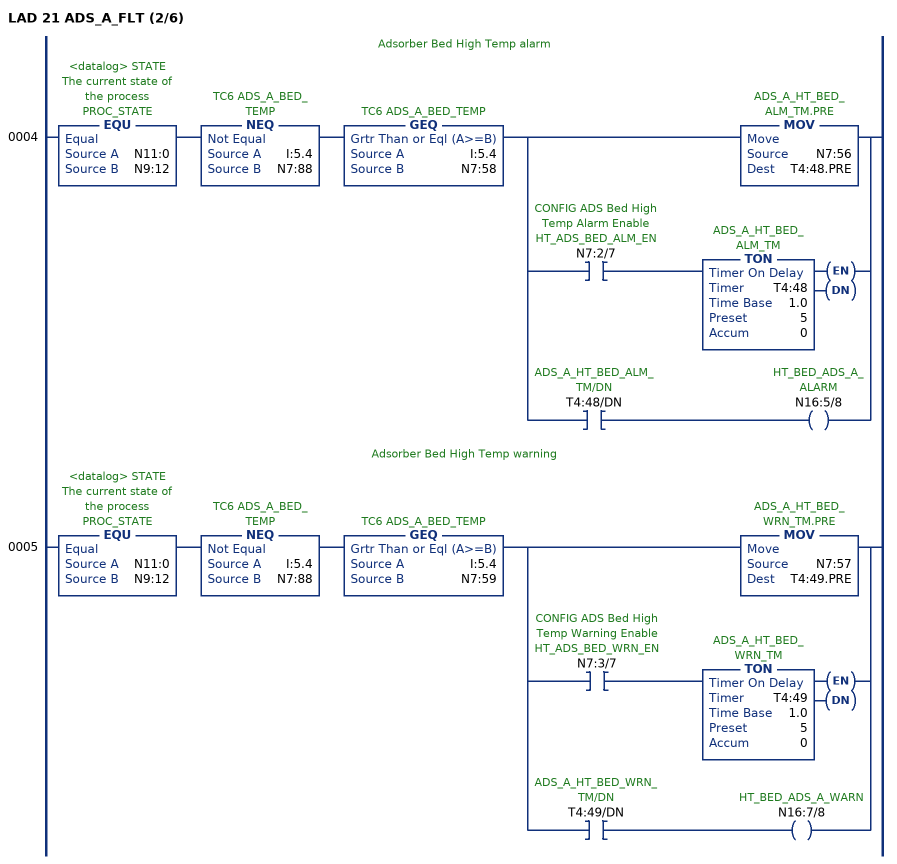
% Rung: 4 %
% Adsorber Bed High Temp alarm %
SOR EQU N11:0 N9:12 NEQ I:5.4 N7:88 GEQ I:5.4 N7:58 BST MOV N7:56 T4:48.PRE NXB XIC N7:2/7 TON T4:48 1.0 5 0 NXB XIC T4:48/DN OTE N16:5/8 BND EOR
%   N11:0  PROC_STATE  "<datalog> STATE The current state of the process" %
%   N9:12  PROC_REGEN_A  "STATE Process Regen A" %
%   I:5.4  ADS_A_BED_TEMP  "TC6" %
%   N7:88  TC_OPEN_SP  "CONFIG TC Open Setpoint" %
%   N7:58  HT_ADS_BED_ALM_SP  "CONFIG ADS Bed High Temp Alarm Setpoint" %
%   N7:56  HT_ADS_BED_ALM_DLY  "CONFIG ADS Bed High Temp Alarm Delay" %
%   T4:48  ADS_A_HT_BED_ALM_TM %
%   N7:2/7  HT_ADS_BED_ALM_EN  "CONFIG ADS Bed High Temp Alarm Enable" %
%   N16:5/8  HT_BED_ADS_A_ALARM %
% Rung: 5 %
% Adsorber Bed High Temp warning %
SOR EQU N11:0 N9:12 NEQ I:5.4 N7:88 GEQ I:5.4 N7:59 BST MOV N7:57 T4:49.PRE NXB XIC N7:3/7 TON T4:49 1.0 5 0 NXB XIC T4:49/DN OTE N16:7/8 BND EOR
%   N11:0  PROC_STATE  "<datalog> STATE The current state of the process" %
%   N9:12  PROC_REGEN_A  "STATE Process Regen A" %
%   I:5.4  ADS_A_BED_TEMP  "TC6" %
%   N7:88  TC_OPEN_SP  "CONFIG TC Open Setpoint" %
%   N7:59  HT_ADS_BED_WRN_SP  "CONFIG ADS Bed High Temp Warning Setpoint" %
%   N7:57  HT_ADS_BED_WRN_DLY  "CONFIG ADS Bed High Temp Warning Delay" %
%   T4:49  ADS_A_HT_BED_WRN_TM %
%   N7:3/7  HT_ADS_BED_WRN_EN  "CONFIG ADS Bed High Temp Warning Enable" %
%   N16:7/8  HT_BED_ADS_A_WARN %

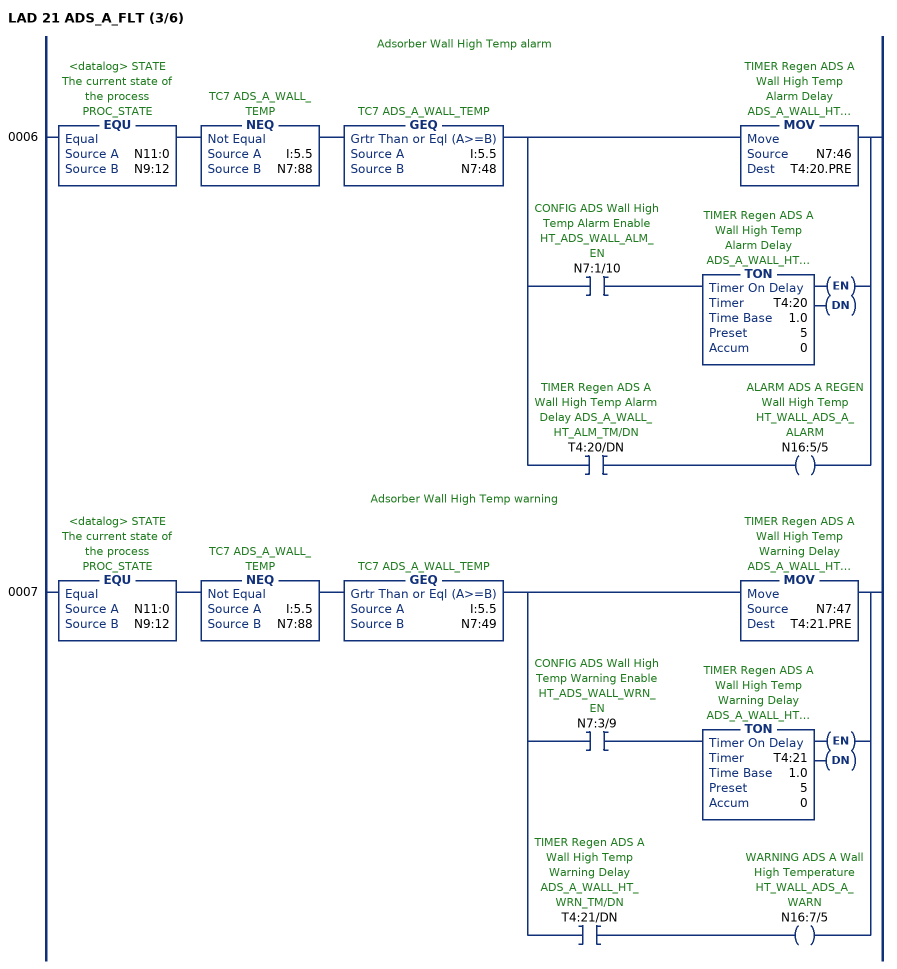
% Rung: 6 %
% Adsorber Wall High Temp alarm %
SOR EQU N11:0 N9:12 NEQ I:5.5 N7:88 GEQ I:5.5 N7:48 BST MOV N7:46 T4:20.PRE NXB XIC N7:1/10 TON T4:20 1.0 5 0 NXB XIC T4:20/DN OTE N16:5/5 BND EOR
%   N11:0  PROC_STATE  "<datalog> STATE The current state of the process" %
%   N9:12  PROC_REGEN_A  "STATE Process Regen A" %
%   I:5.5  ADS_A_WALL_TEMP  "TC7" %
%   N7:88  TC_OPEN_SP  "CONFIG TC Open Setpoint" %
%   N7:48  HT_ADS_WALL_ALM_SP  "CONFIG ADS Wall High Temp Alarm Setpoint" %
%   N7:46  HT_ADS_WALL_ALM_DLY  "CONFIG ADS Wall High Temp Alarm Delay" %
%   T4:20  ADS_A_WALL_HT_ALM_TM  "TIMER Regen ADS A Wall High Temp Alarm Delay" %
%   N7:1/10  HT_ADS_WALL_ALM_EN  "CONFIG ADS Wall High Temp Alarm Enable" %
%   N16:5/5  HT_WALL_ADS_A_ALARM  "ALARM ADS A REGEN Wall High Temp" %
% Rung: 7 %
% Adsorber Wall High Temp warning %
SOR EQU N11:0 N9:12 NEQ I:5.5 N7:88 GEQ I:5.5 N7:49 BST MOV N7:47 T4:21.PRE NXB XIC N7:3/9 TON T4:21 1.0 5 0 NXB XIC T4:21/DN OTE N16:7/5 BND EOR
%   N11:0  PROC_STATE  "<datalog> STATE The current state of the process" %
%   N9:12  PROC_REGEN_A  "STATE Process Regen A" %
%   I:5.5  ADS_A_WALL_TEMP  "TC7" %
%   N7:88  TC_OPEN_SP  "CONFIG TC Open Setpoint" %
%   N7:49  HT_ADS_WALL_WRN_SP  "CONFIG ADS Wall High Temp Warning Setpoint" %
%   N7:47  HT_ADS_WALL_WRN_DLY  "CONFIG ADS Wall High Temp Warning Delay" %
%   T4:21  ADS_A_WALL_HT_WRN_TM  "TIMER Regen ADS A Wall High Temp Warning Delay" %
%   N7:3/9  HT_ADS_WALL_WRN_EN  "CONFIG ADS Wall High Temp Warning Enable" %
%   N16:7/5  HT_WALL_ADS_A_WARN  "WARNING ADS A Wall High Temperature" %

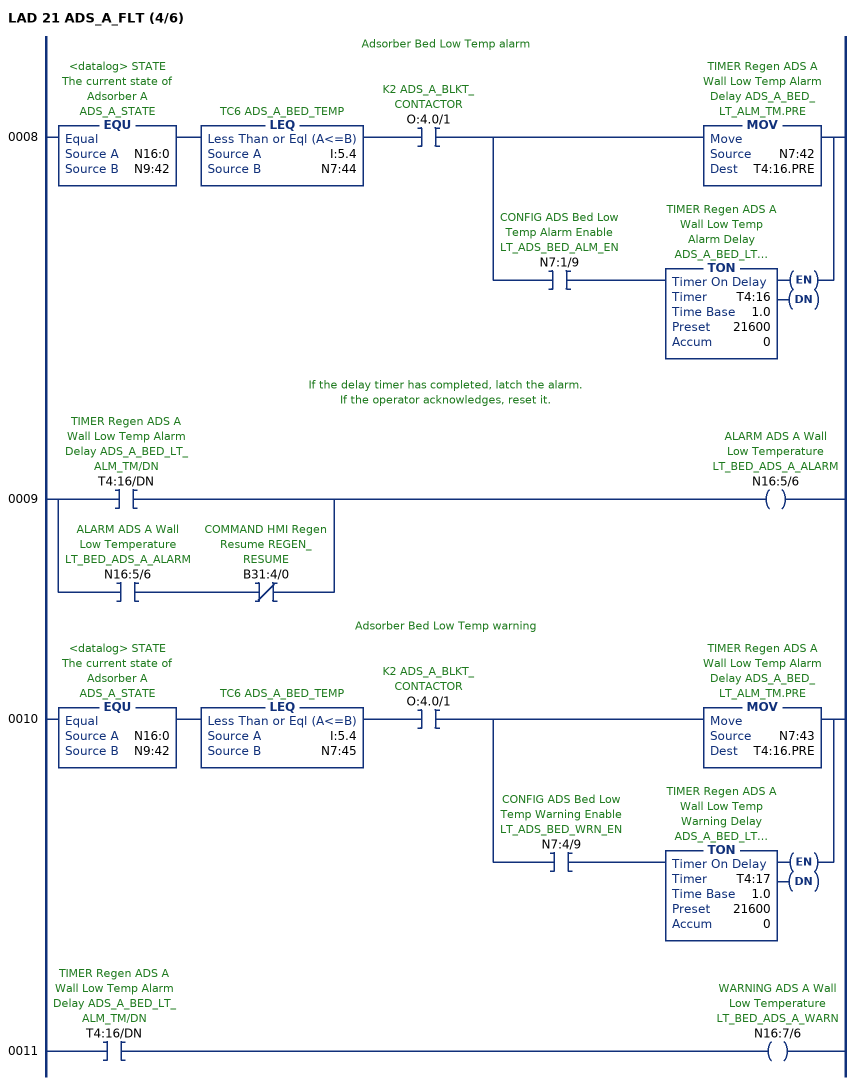
% Rung: 8 %
% Adsorber Bed Low Temp alarm %
SOR EQU N16:0 N9:42 LEQ I:5.4 N7:44 XIC O:4.0/1 BST MOV N7:42 T4:16.PRE NXB XIC N7:1/9 TON T4:16 1.0 21600 0 BND EOR
%   N16:0  ADS_A_STATE  "<datalog> STATE The current state of Adsorber A" %
%   N9:42  ADS_REGEN  "STATE ADS Regen" %
%   I:5.4  ADS_A_BED_TEMP  "TC6" %
%   N7:44  LT_ADS_BED_ALM_SP  "CONFIG ADS Bed Low Temp Alarm Setpoint" %
%   O:4.0/1  ADS_A_BLKT_CONTACTOR  "K2" %
%   N7:42  LT_ADS_BED_ALM_DLY  "CONFIG ADS Bed Low Temp Alarm Delay" %
%   T4:16  ADS_A_BED_LT_ALM_TM  "TIMER Regen ADS A Wall Low Temp Alarm Delay" %
%   N7:1/9  LT_ADS_BED_ALM_EN  "CONFIG ADS Bed Low Temp Alarm Enable" %
% Rung: 9 %
% If the delay timer has completed, latch the alarm.
% If the operator acknowledges, reset it. %
SOR BST XIC T4:16/DN NXB XIC N16:5/6 XIO B31:4/0 BND OTE N16:5/6 EOR
%   T4:16  ADS_A_BED_LT_ALM_TM  "TIMER Regen ADS A Wall Low Temp Alarm Delay" %
%   N16:5/6  LT_BED_ADS_A_ALARM  "ALARM ADS A Wall Low Temperature" %
%   B31:4/0  REGEN_RESUME  "COMMAND HMI Regen Resume" %
% Rung: 10 %
% Adsorber Bed Low Temp warning %
SOR EQU N16:0 N9:42 LEQ I:5.4 N7:45 XIC O:4.0/1 BST MOV N7:43 T4:16.PRE NXB XIC N7:4/9 TON T4:17 1.0 21600 0 BND EOR
%   N16:0  ADS_A_STATE  "<datalog> STATE The current state of Adsorber A" %
%   N9:42  ADS_REGEN  "STATE ADS Regen" %
%   I:5.4  ADS_A_BED_TEMP  "TC6" %
%   N7:45  LT_ADS_BED_WRN_SP  "CONFIG ADS Bed Low Temp Warning Setpoint" %
%   O:4.0/1  ADS_A_BLKT_CONTACTOR  "K2" %
%   N7:43  LT_ADS_BED_WRN_DLY  "CONFIG ADS Bed Low Temp Warning Delay" %
%   T4:16  ADS_A_BED_LT_ALM_TM  "TIMER Regen ADS A Wall Low Temp Alarm Delay" %
%   N7:4/9  LT_ADS_BED_WRN_EN  "CONFIG ADS Bed Low Temp Warning Enable" %
%   T4:17  ADS_A_BED_LT_WRN_TM  "TIMER Regen ADS A Wall Low Temp Warning Delay" %
% Rung: 11 %
SOR XIC T4:16/DN OTE N16:7/6 EOR
%   T4:16  ADS_A_BED_LT_ALM_TM  "TIMER Regen ADS A Wall Low Temp Alarm Delay" %
%   N16:7/6  LT_BED_ADS_A_WARN  "WARNING ADS A Wall Low Temperature" %

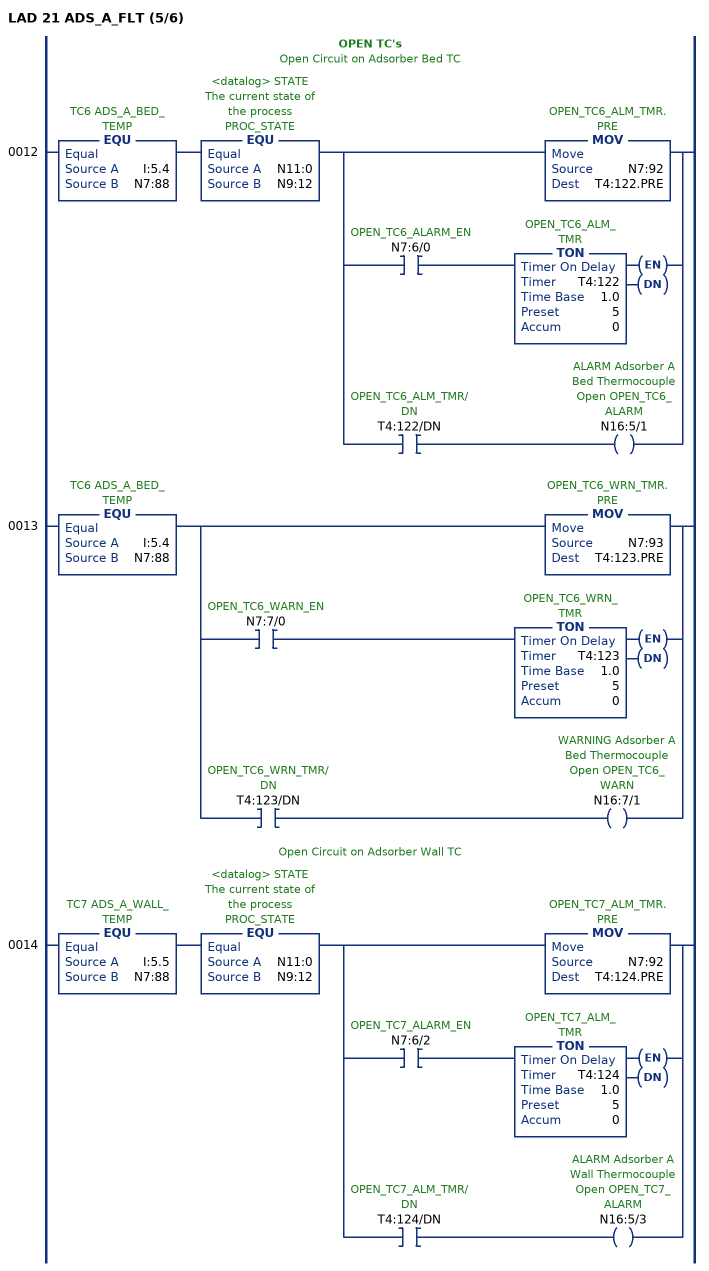
% Rung: 12 %
% TITLE: OPEN TC's %
% Open Circuit on Adsorber Bed TC %
SOR EQU I:5.4 N7:88 EQU N11:0 N9:12 BST MOV N7:92 T4:122.PRE NXB XIC N7:6/0 TON T4:122 1.0 5 0 NXB XIC T4:122/DN OTE N16:5/1 BND EOR
%   I:5.4  ADS_A_BED_TEMP  "TC6" %
%   N7:88  TC_OPEN_SP  "CONFIG TC Open Setpoint" %
%   N11:0  PROC_STATE  "<datalog> STATE The current state of the process" %
%   N9:12  PROC_REGEN_A  "STATE Process Regen A" %
%   N7:92  OPEN_TC_ALM_DLY  "CONFIG TC Open Alarm Delay" %
%   T4:122  OPEN_TC6_ALM_TMR %
%   N7:6/0  OPEN_TC6_ALARM_EN %
%   N16:5/1  OPEN_TC6_ALARM  "ALARM Adsorber A Bed Thermocouple Open" %
% Rung: 13 %
SOR EQU I:5.4 N7:88 BST MOV N7:93 T4:123.PRE NXB XIC N7:7/0 TON T4:123 1.0 5 0 NXB XIC T4:123/DN OTE N16:7/1 BND EOR
%   I:5.4  ADS_A_BED_TEMP  "TC6" %
%   N7:88  TC_OPEN_SP  "CONFIG TC Open Setpoint" %
%   N7:93  OPEN_TC_WRN_DLY  "CONFIG TC Open Warning Delay" %
%   T4:123  OPEN_TC6_WRN_TMR %
%   N7:7/0  OPEN_TC6_WARN_EN %
%   N16:7/1  OPEN_TC6_WARN  "WARNING Adsorber A Bed Thermocouple Open" %
% Rung: 14 %
% Open Circuit on Adsorber Wall TC %
SOR EQU I:5.5 N7:88 EQU N11:0 N9:12 BST MOV N7:92 T4:124.PRE NXB XIC N7:6/2 TON T4:124 1.0 5 0 NXB XIC T4:124/DN OTE N16:5/3 BND EOR
%   I:5.5  ADS_A_WALL_TEMP  "TC7" %
%   N7:88  TC_OPEN_SP  "CONFIG TC Open Setpoint" %
%   N11:0  PROC_STATE  "<datalog> STATE The current state of the process" %
%   N9:12  PROC_REGEN_A  "STATE Process Regen A" %
%   N7:92  OPEN_TC_ALM_DLY  "CONFIG TC Open Alarm Delay" %
%   T4:124  OPEN_TC7_ALM_TMR %
%   N7:6/2  OPEN_TC7_ALARM_EN %
%   N16:5/3  OPEN_TC7_ALARM  "ALARM Adsorber A Wall Thermocouple Open" %

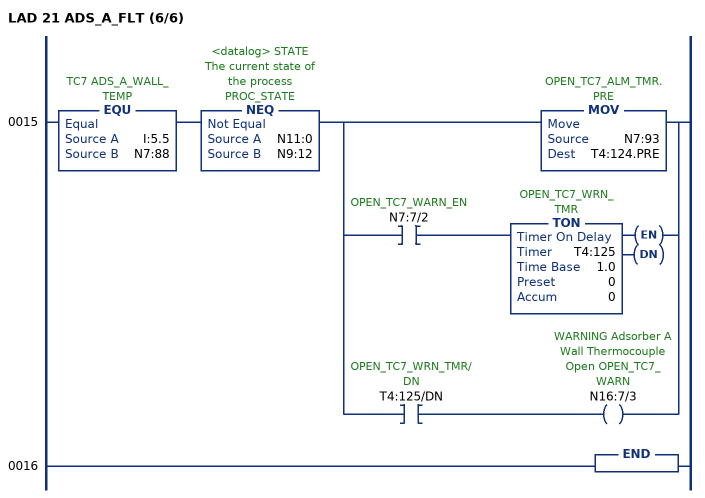
% Rung: 15 %
SOR EQU I:5.5 N7:88 NEQ N11:0 N9:12 BST MOV N7:93 T4:124.PRE NXB XIC N7:7/2 TON T4:125 1.0 0 0 NXB XIC T4:125/DN OTE N16:7/3 BND EOR
%   I:5.5  ADS_A_WALL_TEMP  "TC7" %
%   N7:88  TC_OPEN_SP  "CONFIG TC Open Setpoint" %
%   N11:0  PROC_STATE  "<datalog> STATE The current state of the process" %
%   N9:12  PROC_REGEN_A  "STATE Process Regen A" %
%   N7:93  OPEN_TC_WRN_DLY  "CONFIG TC Open Warning Delay" %
%   T4:124  OPEN_TC7_ALM_TMR %
%   N7:7/2  OPEN_TC7_WARN_EN %
%   T4:125  OPEN_TC7_WRN_TMR %
%   N16:7/3  OPEN_TC7_WARN  "WARNING Adsorber A Wall Thermocouple Open" %
% Rung: 16 %
SOR END EOR

LADDER 22 "ADS_B"    % Controld Adsorber B %
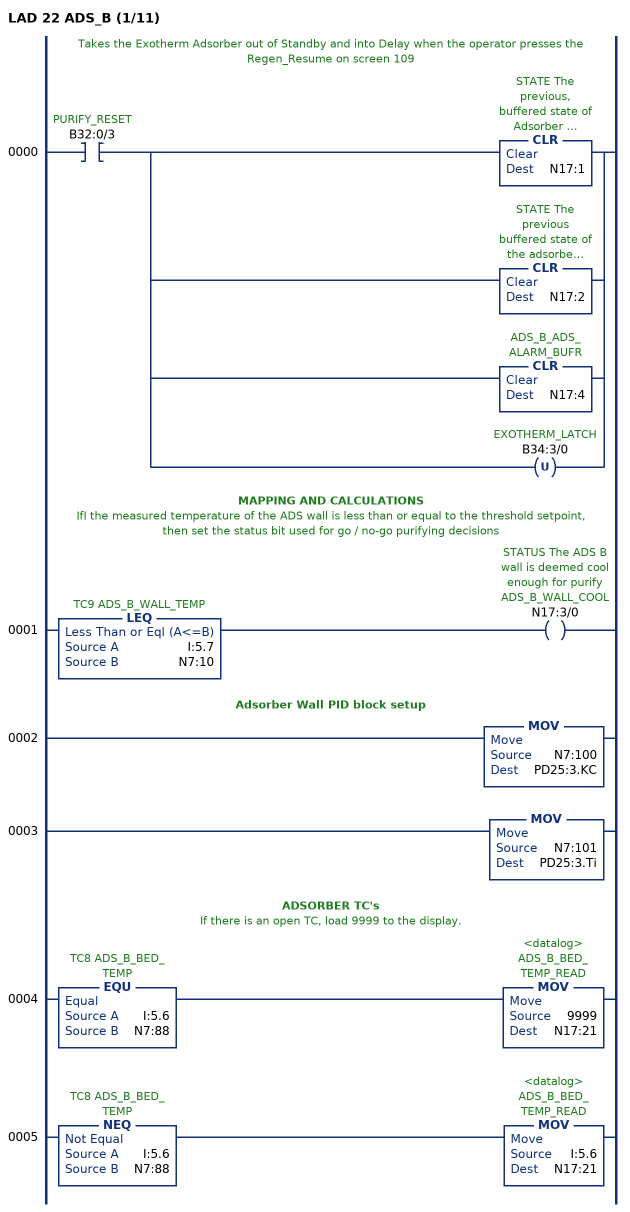
% Rung: 0 %
% Takes the Exotherm Adsorber out of Standby and into Delay when the operator presses the Regen_Resume on screen 109 %
SOR XIC B32:0/3 BST CLR N17:1 NXB CLR N17:2 NXB CLR N17:4 NXB OTU B34:3/0 BND EOR
%   B32:0/3  PURIFY_RESET %
%   N17:1  ADS_B_STANDBY_BUFFER  "STATE The previous, buffered state of Adsorber B" %
%   N17:2  ADS_B_SYS_ALARM_BUFR  "STATE The previous buffered state of the adsorber when the alarm occured" %
%   N17:4  ADS_B_ADS_ALARM_BUFR %
%   B34:3/0  EXOTHERM_LATCH %
% Rung: 1 %
% TITLE: MAPPING AND CALCULATIONS %
% IfI the measured temperature of the ADS wall is less than or equal to the threshold setpoint, then set the status bit used for go / no-go purifying decisions %
SOR LEQ I:5.7 N7:10 OTE N17:3/0 EOR
%   I:5.7  ADS_B_WALL_TEMP  "TC9" %
%   N7:10  ADS_WALL_TEMP_COOL  "CONFIG The temp at which the adsorber wall is deemed to be cool enough to purify" %
%   N17:3/0  ADS_B_WALL_COOL  "STATUS The ADS B wall is deemed cool enough for purify" %
% Rung: 2 %
% TITLE: Adsorber Wall PID block setup %
SOR MOV N7:100 PD25:3.KC EOR
%   N7:100  BLANKET_P  "CONFIG Blanket Proportional Gain" %
% Rung: 3 %
SOR MOV N7:101 PD25:3.Ti EOR
%   N7:101  BLANKET_I  "CONFIG Blanket Integral Gain" %
% Rung: 4 %
% TITLE: ADSORBER TC's %
% If there is an open TC, load 9999 to the display. %
SOR EQU I:5.6 N7:88 MOV 9999 N17:21 EOR
%   I:5.6  ADS_B_BED_TEMP  "TC8" %
%   N7:88  TC_OPEN_SP  "CONFIG TC Open Setpoint" %
%   N17:21  ADS_B_BED_TEMP_READ  "<datalog>" %
% Rung: 5 %
SOR NEQ I:5.6 N7:88 MOV I:5.6 N17:21 EOR
%   I:5.6  ADS_B_BED_TEMP  "TC8" %
%   N7:88  TC_OPEN_SP  "CONFIG TC Open Setpoint" %
%   N17:21  ADS_B_BED_TEMP_READ  "<datalog>" %

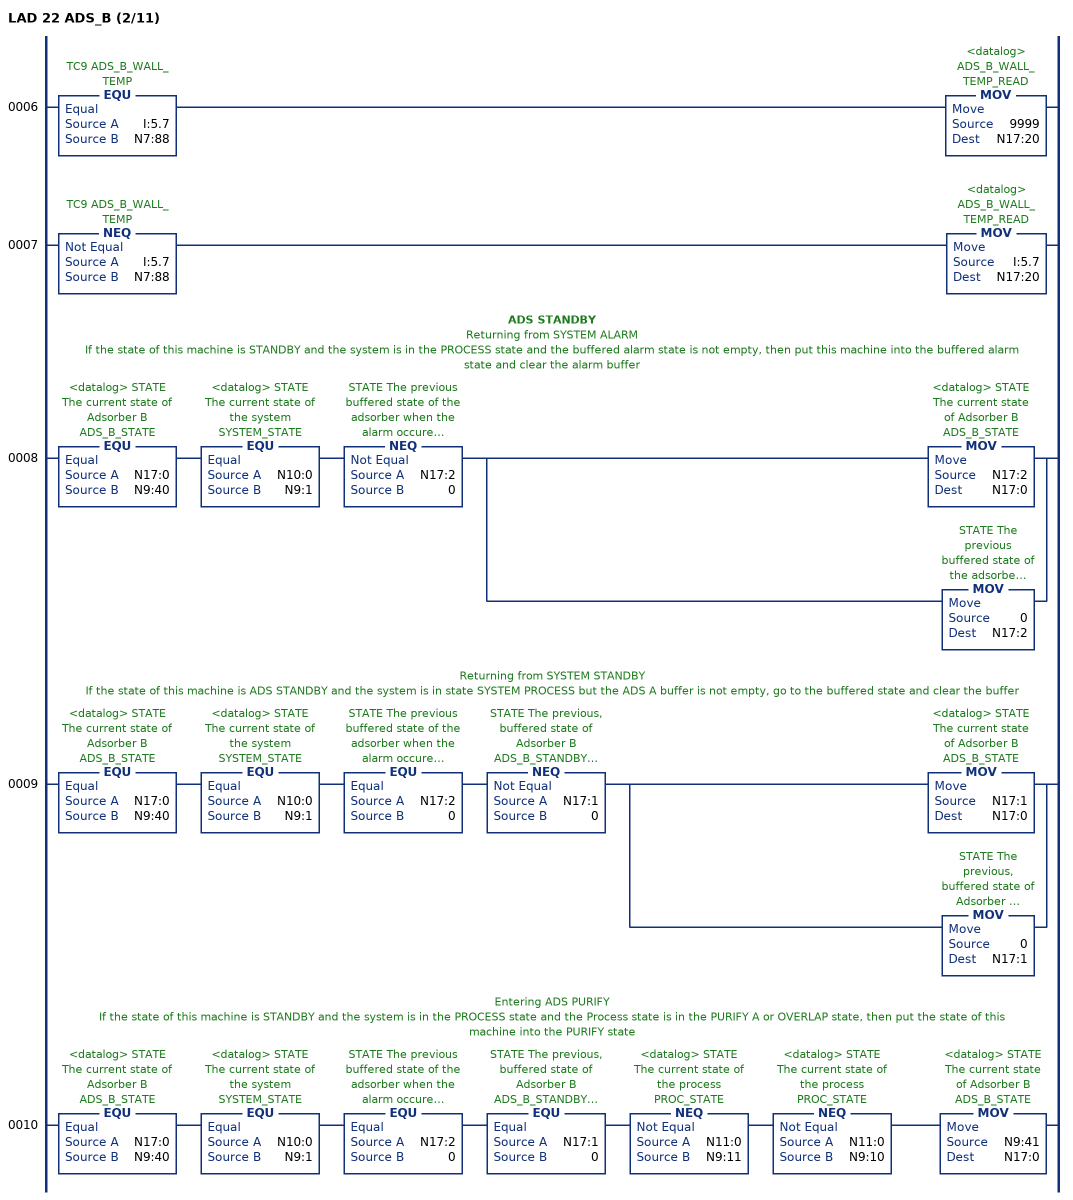
% Rung: 6 %
SOR EQU I:5.7 N7:88 MOV 9999 N17:20 EOR
%   I:5.7  ADS_B_WALL_TEMP  "TC9" %
%   N7:88  TC_OPEN_SP  "CONFIG TC Open Setpoint" %
%   N17:20  ADS_B_WALL_TEMP_READ  "<datalog>" %
% Rung: 7 %
SOR NEQ I:5.7 N7:88 MOV I:5.7 N17:20 EOR
%   I:5.7  ADS_B_WALL_TEMP  "TC9" %
%   N7:88  TC_OPEN_SP  "CONFIG TC Open Setpoint" %
%   N17:20  ADS_B_WALL_TEMP_READ  "<datalog>" %
% Rung: 8 %
% TITLE: ADS STANDBY %
% Returning from SYSTEM ALARM
% If the state of this machine is STANDBY and the system is in the PROCESS state and the buffered alarm state is not empty, then put this machine into the buffered alarm state and clear the alarm buffer %
SOR EQU N17:0 N9:40 EQU N10:0 N9:1 NEQ N17:2 0 BST MOV N17:2 N17:0 NXB MOV 0 N17:2 BND EOR
%   N17:0  ADS_B_STATE  "<datalog> STATE The current state of Adsorber B" %
%   N9:40  ADS_STANDBY  "STATE ADS Standby" %
%   N10:0  SYSTEM_STATE  "<datalog> STATE The current state of the system" %
%   N9:1  SYSTEM_PROCESS  "STATE System Process" %
%   N17:2  ADS_B_SYS_ALARM_BUFR  "STATE The previous buffered state of the adsorber when the alarm occured" %
% Rung: 9 %
% Returning from SYSTEM STANDBY
% If the state of this machine is ADS STANDBY and the system is in state SYSTEM PROCESS but the ADS A buffer is not empty, go to the buffered state and clear the buffer %
SOR EQU N17:0 N9:40 EQU N10:0 N9:1 EQU N17:2 0 NEQ N17:1 0 BST MOV N17:1 N17:0 NXB MOV 0 N17:1 BND EOR
%   N17:0  ADS_B_STATE  "<datalog> STATE The current state of Adsorber B" %
%   N9:40  ADS_STANDBY  "STATE ADS Standby" %
%   N10:0  SYSTEM_STATE  "<datalog> STATE The current state of the system" %
%   N9:1  SYSTEM_PROCESS  "STATE System Process" %
%   N17:2  ADS_B_SYS_ALARM_BUFR  "STATE The previous buffered state of the adsorber when the alarm occured" %
%   N17:1  ADS_B_STANDBY_BUFFER  "STATE The previous, buffered state of Adsorber B" %
% Rung: 10 %
% Entering ADS PURIFY
% If the state of this machine is STANDBY and the system is in the PROCESS state and the Process state is in the PURIFY A or OVERLAP state, then put the state of this machine into the PURIFY state %
SOR EQU N17:0 N9:40 EQU N10:0 N9:1 EQU N17:2 0 EQU N17:1 0 NEQ N11:0 N9:11 NEQ N11:0 N9:10 MOV N9:41 N17:0 EOR
%   N17:0  ADS_B_STATE  "<datalog> STATE The current state of Adsorber B" %
%   N9:40  ADS_STANDBY  "STATE ADS Standby" %
%   N10:0  SYSTEM_STATE  "<datalog> STATE The current state of the system" %
%   N9:1  SYSTEM_PROCESS  "STATE System Process" %
%   N17:2  ADS_B_SYS_ALARM_BUFR  "STATE The previous buffered state of the adsorber when the alarm occured" %
%   N17:1  ADS_B_STANDBY_BUFFER  "STATE The previous, buffered state of Adsorber B" %
%   N11:0  PROC_STATE  "<datalog> STATE The current state of the process" %
%   N9:11  PROC_REGEN_B  "STATE Process Regen B" %
%   N9:10  PROCESS_STANDBY  "STATE Process Standby" %
%   N9:41  ADS_PURIFY  "STATE ADS Purify" %

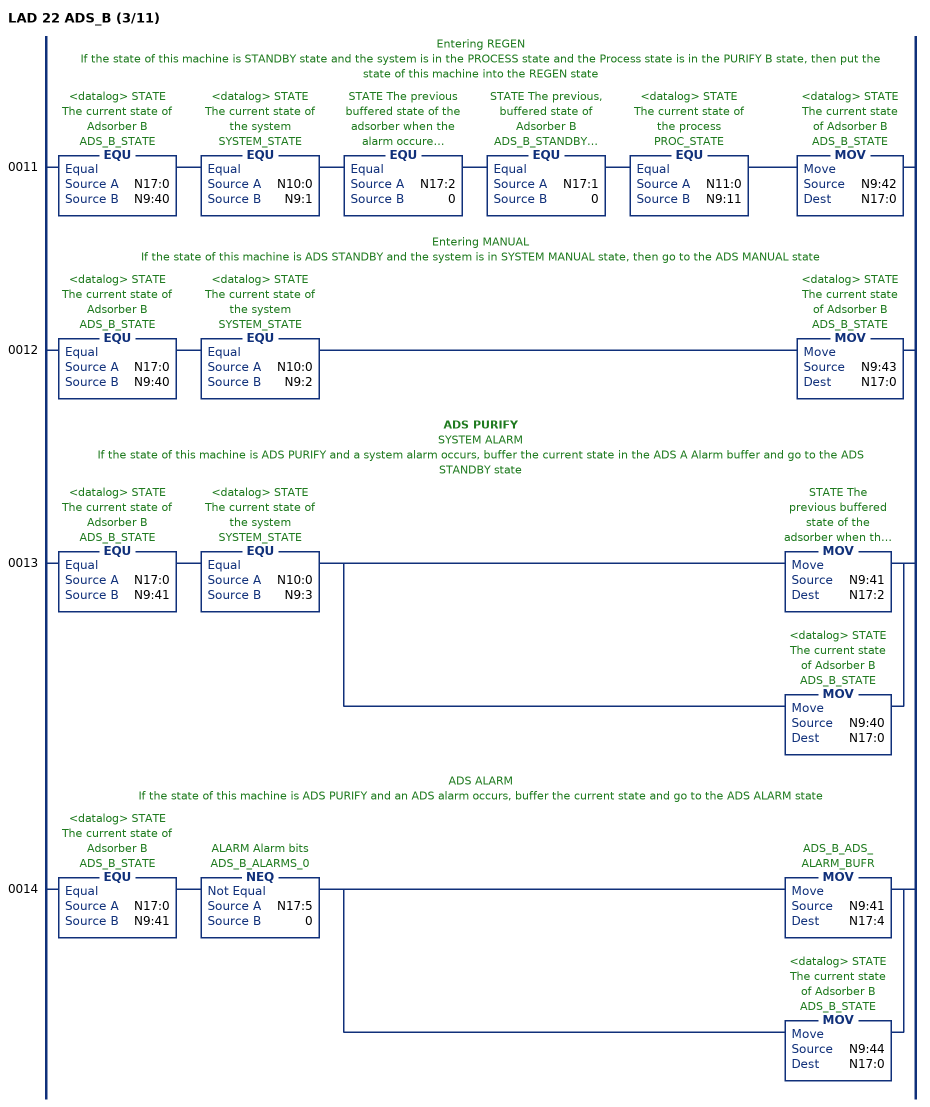
% Rung: 11 %
% Entering REGEN
% If the state of this machine is STANDBY state and the system is in the PROCESS state and the Process state is in the PURIFY B state, then put the state of this machine into the REGEN state %
SOR EQU N17:0 N9:40 EQU N10:0 N9:1 EQU N17:2 0 EQU N17:1 0 EQU N11:0 N9:11 MOV N9:42 N17:0 EOR
%   N17:0  ADS_B_STATE  "<datalog> STATE The current state of Adsorber B" %
%   N9:40  ADS_STANDBY  "STATE ADS Standby" %
%   N10:0  SYSTEM_STATE  "<datalog> STATE The current state of the system" %
%   N9:1  SYSTEM_PROCESS  "STATE System Process" %
%   N17:2  ADS_B_SYS_ALARM_BUFR  "STATE The previous buffered state of the adsorber when the alarm occured" %
%   N17:1  ADS_B_STANDBY_BUFFER  "STATE The previous, buffered state of Adsorber B" %
%   N11:0  PROC_STATE  "<datalog> STATE The current state of the process" %
%   N9:11  PROC_REGEN_B  "STATE Process Regen B" %
%   N9:42  ADS_REGEN  "STATE ADS Regen" %
% Rung: 12 %
% Entering MANUAL
% If the state of this machine is ADS STANDBY and the system is in SYSTEM MANUAL state, then go to the ADS MANUAL state %
SOR EQU N17:0 N9:40 EQU N10:0 N9:2 MOV N9:43 N17:0 EOR
%   N17:0  ADS_B_STATE  "<datalog> STATE The current state of Adsorber B" %
%   N9:40  ADS_STANDBY  "STATE ADS Standby" %
%   N10:0  SYSTEM_STATE  "<datalog> STATE The current state of the system" %
%   N9:2  SYSTEM_MANUAL  "STATE System Manual" %
%   N9:43  ADS_MANUAL  "STATE ADS Manual" %
% Rung: 13 %
% TITLE: ADS PURIFY %
% SYSTEM ALARM
% If the state of this machine is ADS PURIFY and a system alarm occurs, buffer the current state in the ADS A Alarm buffer and go to the ADS STANDBY state %
SOR EQU N17:0 N9:41 EQU N10:0 N9:3 BST MOV N9:41 N17:2 NXB MOV N9:40 N17:0 BND EOR
%   N17:0  ADS_B_STATE  "<datalog> STATE The current state of Adsorber B" %
%   N9:41  ADS_PURIFY  "STATE ADS Purify" %
%   N10:0  SYSTEM_STATE  "<datalog> STATE The current state of the system" %
%   N9:3  SYSTEM_ALARM  "STATE System Alarm" %
%   N17:2  ADS_B_SYS_ALARM_BUFR  "STATE The previous buffered state of the adsorber when the alarm occured" %
%   N9:40  ADS_STANDBY  "STATE ADS Standby" %
% Rung: 14 %
% ADS ALARM
% If the state of this machine is ADS PURIFY and an ADS alarm occurs, buffer the current state and go to the ADS ALARM state %
SOR EQU N17:0 N9:41 NEQ N17:5 0 BST MOV N9:41 N17:4 NXB MOV N9:44 N17:0 BND EOR
%   N17:0  ADS_B_STATE  "<datalog> STATE The current state of Adsorber B" %
%   N9:41  ADS_PURIFY  "STATE ADS Purify" %
%   N17:5  ADS_B_ALARMS_0  "ALARM Alarm bits" %
%   N17:4  ADS_B_ADS_ALARM_BUFR %
%   N9:44  ADS_ALARM  "STATE ADS Alarm" %

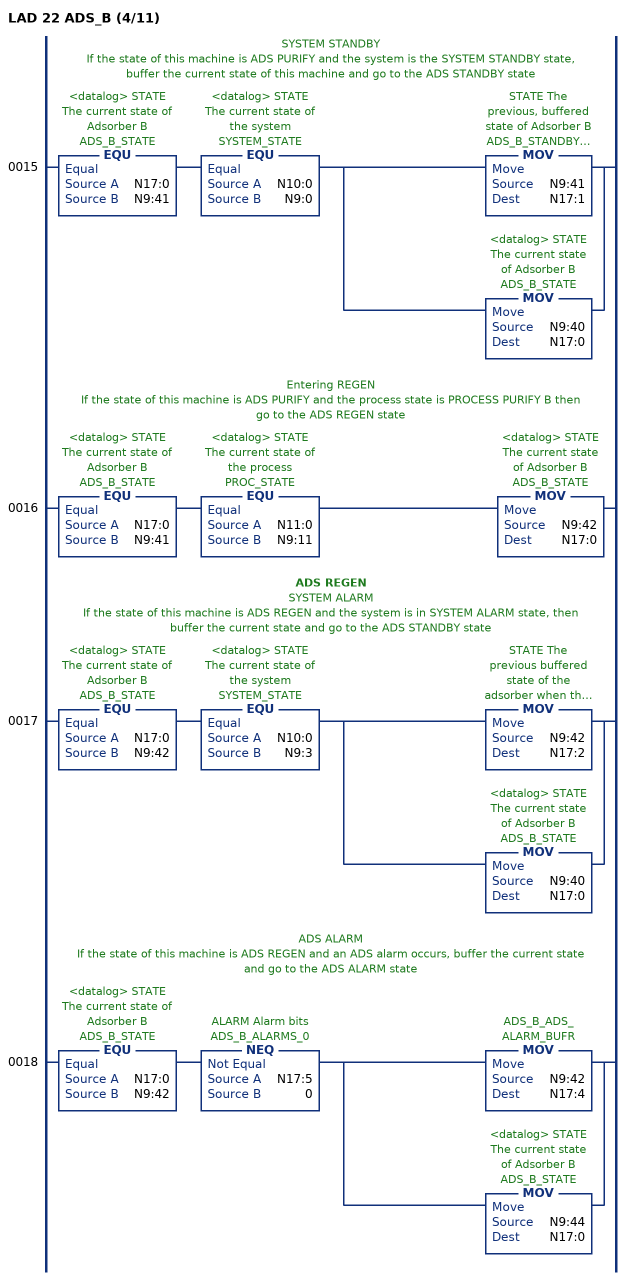
% Rung: 15 %
% SYSTEM STANDBY
% If the state of this machine is ADS PURIFY and the system is the SYSTEM STANDBY state, buffer the current state of this machine and go to the ADS STANDBY state %
SOR EQU N17:0 N9:41 EQU N10:0 N9:0 BST MOV N9:41 N17:1 NXB MOV N9:40 N17:0 BND EOR
%   N17:0  ADS_B_STATE  "<datalog> STATE The current state of Adsorber B" %
%   N9:41  ADS_PURIFY  "STATE ADS Purify" %
%   N10:0  SYSTEM_STATE  "<datalog> STATE The current state of the system" %
%   N9:0  SYSTEM_STANDBY  "STATE System Standby" %
%   N17:1  ADS_B_STANDBY_BUFFER  "STATE The previous, buffered state of Adsorber B" %
%   N9:40  ADS_STANDBY  "STATE ADS Standby" %
% Rung: 16 %
% Entering REGEN
% If the state of this machine is ADS PURIFY and the process state is PROCESS PURIFY B then go to the ADS REGEN state %
SOR EQU N17:0 N9:41 EQU N11:0 N9:11 MOV N9:42 N17:0 EOR
%   N17:0  ADS_B_STATE  "<datalog> STATE The current state of Adsorber B" %
%   N9:41  ADS_PURIFY  "STATE ADS Purify" %
%   N11:0  PROC_STATE  "<datalog> STATE The current state of the process" %
%   N9:11  PROC_REGEN_B  "STATE Process Regen B" %
%   N9:42  ADS_REGEN  "STATE ADS Regen" %
% Rung: 17 %
% TITLE: ADS REGEN %
% SYSTEM ALARM
% If the state of this machine is ADS REGEN and the system is in SYSTEM ALARM state, then buffer the current state and go to the ADS STANDBY state %
SOR EQU N17:0 N9:42 EQU N10:0 N9:3 BST MOV N9:42 N17:2 NXB MOV N9:40 N17:0 BND EOR
%   N17:0  ADS_B_STATE  "<datalog> STATE The current state of Adsorber B" %
%   N9:42  ADS_REGEN  "STATE ADS Regen" %
%   N10:0  SYSTEM_STATE  "<datalog> STATE The current state of the system" %
%   N9:3  SYSTEM_ALARM  "STATE System Alarm" %
%   N17:2  ADS_B_SYS_ALARM_BUFR  "STATE The previous buffered state of the adsorber when the alarm occured" %
%   N9:40  ADS_STANDBY  "STATE ADS Standby" %
% Rung: 18 %
% ADS ALARM
% If the state of this machine is ADS REGEN and an ADS alarm occurs, buffer the current state and go to the ADS ALARM state %
SOR EQU N17:0 N9:42 NEQ N17:5 0 BST MOV N9:42 N17:4 NXB MOV N9:44 N17:0 BND EOR
%   N17:0  ADS_B_STATE  "<datalog> STATE The current state of Adsorber B" %
%   N9:42  ADS_REGEN  "STATE ADS Regen" %
%   N17:5  ADS_B_ALARMS_0  "ALARM Alarm bits" %
%   N17:4  ADS_B_ADS_ALARM_BUFR %
%   N9:44  ADS_ALARM  "STATE ADS Alarm" %

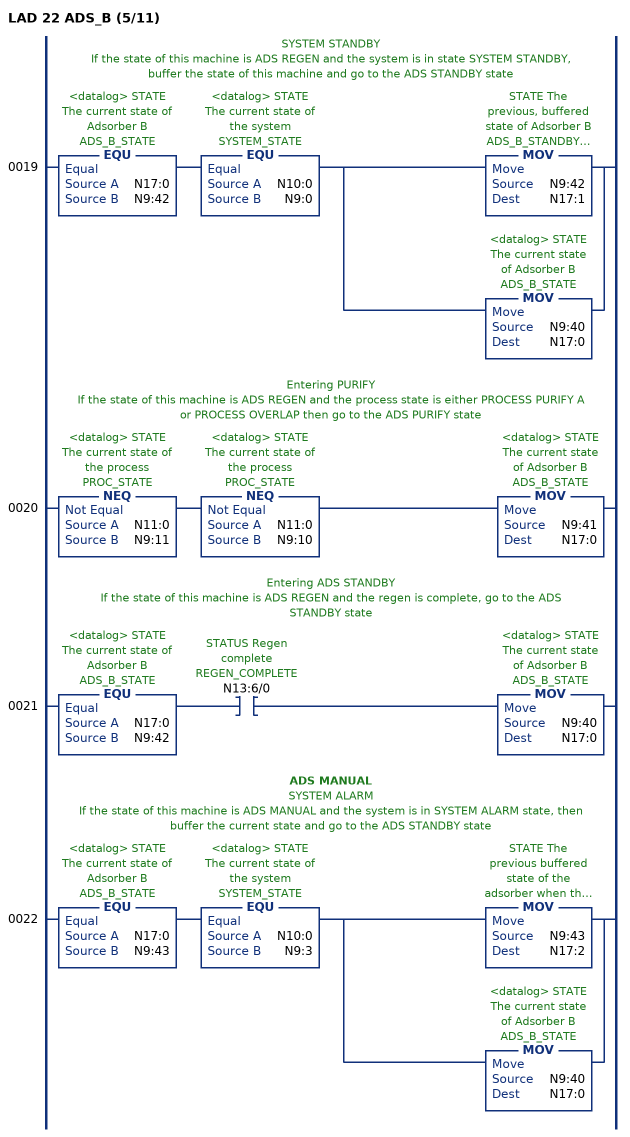
% Rung: 19 %
% SYSTEM STANDBY
% If the state of this machine is ADS REGEN and the system is in state SYSTEM STANDBY, buffer the state of this machine and go to the ADS STANDBY state %
SOR EQU N17:0 N9:42 EQU N10:0 N9:0 BST MOV N9:42 N17:1 NXB MOV N9:40 N17:0 BND EOR
%   N17:0  ADS_B_STATE  "<datalog> STATE The current state of Adsorber B" %
%   N9:42  ADS_REGEN  "STATE ADS Regen" %
%   N10:0  SYSTEM_STATE  "<datalog> STATE The current state of the system" %
%   N9:0  SYSTEM_STANDBY  "STATE System Standby" %
%   N17:1  ADS_B_STANDBY_BUFFER  "STATE The previous, buffered state of Adsorber B" %
%   N9:40  ADS_STANDBY  "STATE ADS Standby" %
% Rung: 20 %
% Entering PURIFY
% If the state of this machine is ADS REGEN and the process state is either PROCESS PURIFY A or PROCESS OVERLAP then go to the ADS PURIFY state %
SOR NEQ N11:0 N9:11 NEQ N11:0 N9:10 MOV N9:41 N17:0 EOR
%   N11:0  PROC_STATE  "<datalog> STATE The current state of the process" %
%   N9:11  PROC_REGEN_B  "STATE Process Regen B" %
%   N9:10  PROCESS_STANDBY  "STATE Process Standby" %
%   N9:41  ADS_PURIFY  "STATE ADS Purify" %
%   N17:0  ADS_B_STATE  "<datalog> STATE The current state of Adsorber B" %
% Rung: 21 %
% Entering ADS STANDBY
% If the state of this machine is ADS REGEN and the regen is complete, go to the ADS STANDBY state %
SOR EQU N17:0 N9:42 XIC N13:6/0 MOV N9:40 N17:0 EOR
%   N17:0  ADS_B_STATE  "<datalog> STATE The current state of Adsorber B" %
%   N9:42  ADS_REGEN  "STATE ADS Regen" %
%   N13:6/0  REGEN_COMPLETE  "STATUS Regen complete" %
%   N9:40  ADS_STANDBY  "STATE ADS Standby" %
% Rung: 22 %
% TITLE: ADS MANUAL %
% SYSTEM ALARM
% If the state of this machine is ADS MANUAL and the system is in SYSTEM ALARM state, then buffer the current state and go to the ADS STANDBY state %
SOR EQU N17:0 N9:43 EQU N10:0 N9:3 BST MOV N9:43 N17:2 NXB MOV N9:40 N17:0 BND EOR
%   N17:0  ADS_B_STATE  "<datalog> STATE The current state of Adsorber B" %
%   N9:43  ADS_MANUAL  "STATE ADS Manual" %
%   N10:0  SYSTEM_STATE  "<datalog> STATE The current state of the system" %
%   N9:3  SYSTEM_ALARM  "STATE System Alarm" %
%   N17:2  ADS_B_SYS_ALARM_BUFR  "STATE The previous buffered state of the adsorber when the alarm occured" %
%   N9:40  ADS_STANDBY  "STATE ADS Standby" %

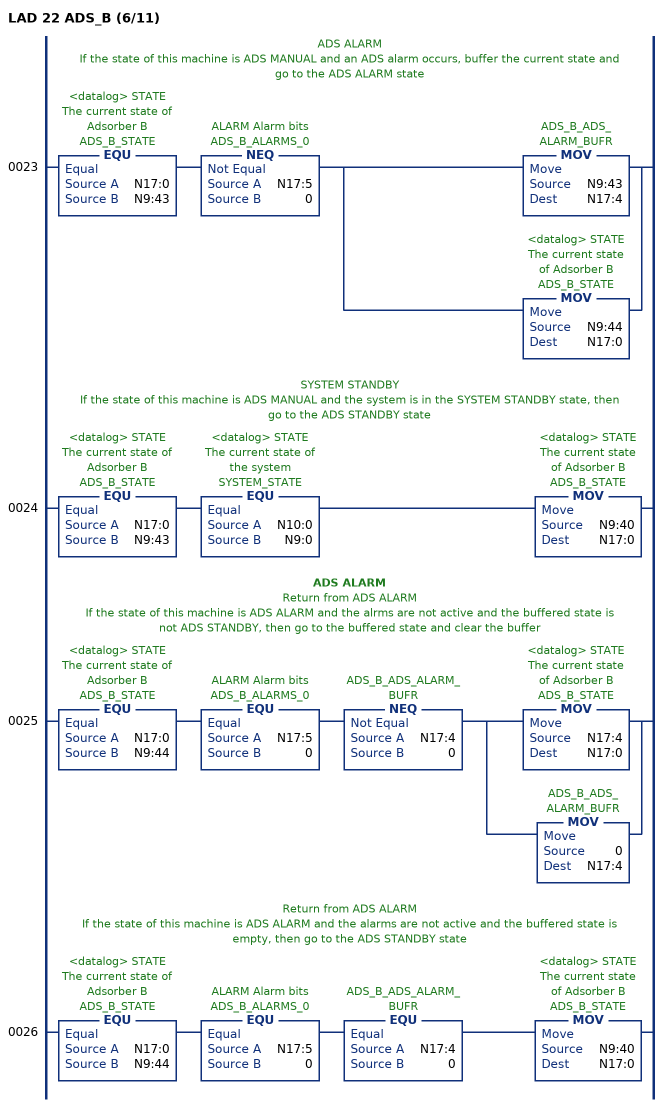
% Rung: 23 %
% ADS ALARM
% If the state of this machine is ADS MANUAL and an ADS alarm occurs, buffer the current state and go to the ADS ALARM state %
SOR EQU N17:0 N9:43 NEQ N17:5 0 BST MOV N9:43 N17:4 NXB MOV N9:44 N17:0 BND EOR
%   N17:0  ADS_B_STATE  "<datalog> STATE The current state of Adsorber B" %
%   N9:43  ADS_MANUAL  "STATE ADS Manual" %
%   N17:5  ADS_B_ALARMS_0  "ALARM Alarm bits" %
%   N17:4  ADS_B_ADS_ALARM_BUFR %
%   N9:44  ADS_ALARM  "STATE ADS Alarm" %
% Rung: 24 %
% SYSTEM STANDBY
% If the state of this machine is ADS MANUAL and the system is in the SYSTEM STANDBY state, then go to the ADS STANDBY state %
SOR EQU N17:0 N9:43 EQU N10:0 N9:0 MOV N9:40 N17:0 EOR
%   N17:0  ADS_B_STATE  "<datalog> STATE The current state of Adsorber B" %
%   N9:43  ADS_MANUAL  "STATE ADS Manual" %
%   N10:0  SYSTEM_STATE  "<datalog> STATE The current state of the system" %
%   N9:0  SYSTEM_STANDBY  "STATE System Standby" %
%   N9:40  ADS_STANDBY  "STATE ADS Standby" %
% Rung: 25 %
% TITLE: ADS ALARM %
% Return from ADS ALARM
% If the state of this machine is ADS ALARM and the alrms are not active and the buffered state is not ADS STANDBY, then go to the buffered state and clear the buffer %
SOR EQU N17:0 N9:44 EQU N17:5 0 NEQ N17:4 0 BST MOV N17:4 N17:0 NXB MOV 0 N17:4 BND EOR
%   N17:0  ADS_B_STATE  "<datalog> STATE The current state of Adsorber B" %
%   N9:44  ADS_ALARM  "STATE ADS Alarm" %
%   N17:5  ADS_B_ALARMS_0  "ALARM Alarm bits" %
%   N17:4  ADS_B_ADS_ALARM_BUFR %
% Rung: 26 %
% Return from ADS ALARM
% If the state of this machine is ADS ALARM and the alarms are not active and the buffered state is empty, then go to the ADS STANDBY state %
SOR EQU N17:0 N9:44 EQU N17:5 0 EQU N17:4 0 MOV N9:40 N17:0 EOR
%   N17:0  ADS_B_STATE  "<datalog> STATE The current state of Adsorber B" %
%   N9:44  ADS_ALARM  "STATE ADS Alarm" %
%   N17:5  ADS_B_ALARMS_0  "ALARM Alarm bits" %
%   N17:4  ADS_B_ADS_ALARM_BUFR %
%   N9:40  ADS_STANDBY  "STATE ADS Standby" %

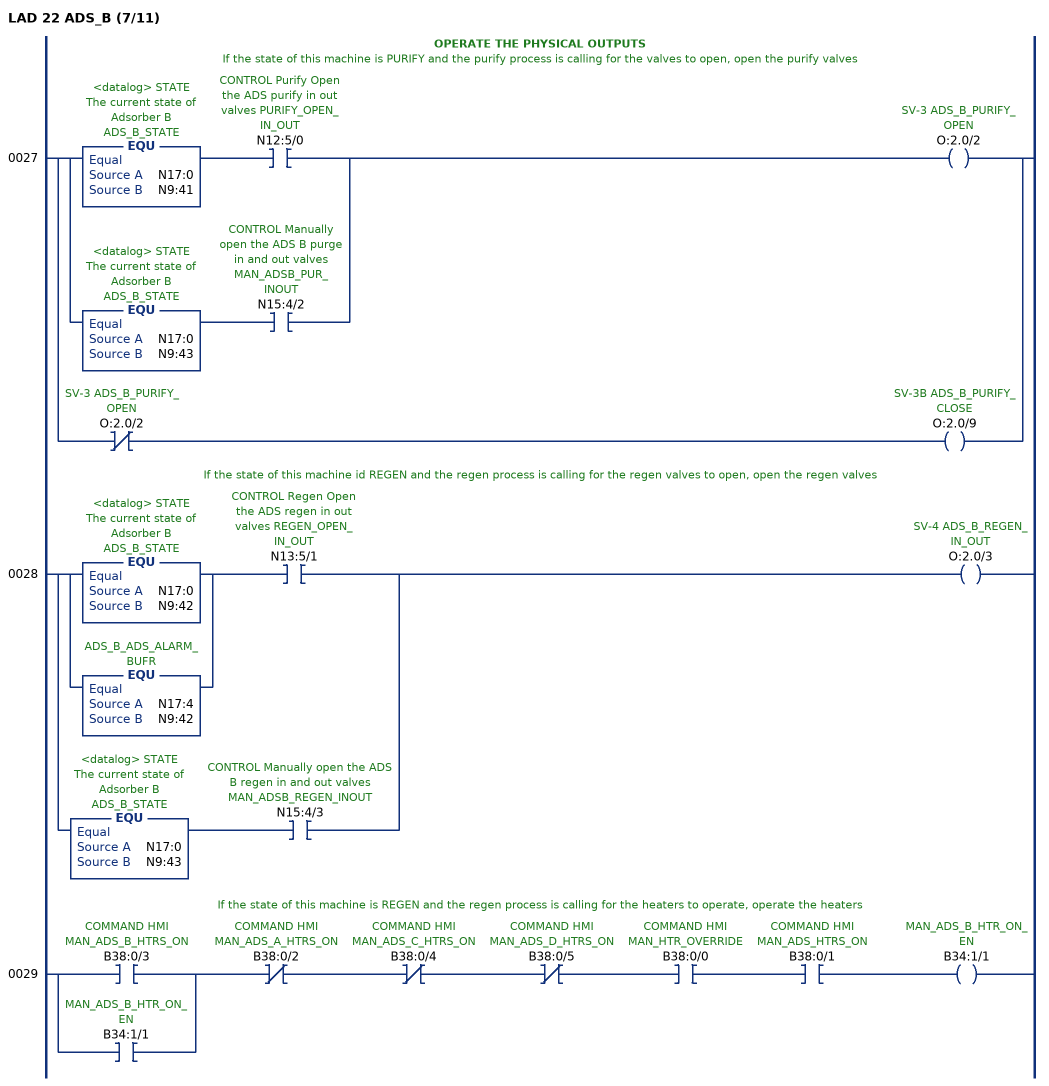
% Rung: 27 %
% TITLE: OPERATE THE PHYSICAL OUTPUTS %
% If the state of this machine is PURIFY and the purify process is calling for the valves to open, open the purify valves %
SOR BST BST EQU N17:0 N9:41 XIC N12:5/0 NXB EQU N17:0 N9:43 XIC N15:4/2 BND OTE O:2.0/2 NXB XIO O:2.0/2 OTE O:2.0/9 BND EOR
%   N17:0  ADS_B_STATE  "<datalog> STATE The current state of Adsorber B" %
%   N9:41  ADS_PURIFY  "STATE ADS Purify" %
%   N12:5/0  PURIFY_OPEN_IN_OUT  "CONTROL Purify Open the ADS purify in out valves" %
%   N9:43  ADS_MANUAL  "STATE ADS Manual" %
%   N15:4/2  MAN_ADSB_PUR_INOUT  "CONTROL Manually open the ADS B purge in and out valves" %
%   O:2.0/2  ADS_B_PURIFY_OPEN  "SV-3" %
%   O:2.0/9  ADS_B_PURIFY_CLOSE  "SV-3B" %
% Rung: 28 %
% If the state of this machine id REGEN and the regen process is calling for the regen valves to open, open the regen valves %
SOR BST BST EQU N17:0 N9:42 NXB EQU N17:4 N9:42 BND XIC N13:5/1 NXB EQU N17:0 N9:43 XIC N15:4/3 BND OTE O:2.0/3 EOR
%   N17:0  ADS_B_STATE  "<datalog> STATE The current state of Adsorber B" %
%   N9:42  ADS_REGEN  "STATE ADS Regen" %
%   N17:4  ADS_B_ADS_ALARM_BUFR %
%   N13:5/1  REGEN_OPEN_IN_OUT  "CONTROL Regen Open the ADS regen in out valves" %
%   N9:43  ADS_MANUAL  "STATE ADS Manual" %
%   N15:4/3  MAN_ADSB_REGEN_INOUT  "CONTROL Manually open the ADS B regen in and out valves" %
%   O:2.0/3  ADS_B_REGEN_IN_OUT  "SV-4" %
% Rung: 29 %
% If the state of this machine is REGEN and the regen process is calling for the heaters to operate, operate the heaters %
SOR BST XIC B38:0/3 NXB XIC B34:1/1 BND XIO B38:0/2 XIO B38:0/4 XIO B38:0/5 XIC B38:0/0 XIC B38:0/1 OTE B34:1/1 EOR
%   B38:0/3  MAN_ADS_B_HTRS_ON  "COMMAND HMI" %
%   B34:1/1  MAN_ADS_B_HTR_ON_EN %
%   B38:0/2  MAN_ADS_A_HTRS_ON  "COMMAND HMI" %
%   B38:0/4  MAN_ADS_C_HTRS_ON  "COMMAND HMI" %
%   B38:0/5  MAN_ADS_D_HTRS_ON  "COMMAND HMI" %
%   B38:0/0  MAN_HTR_OVERRIDE  "COMMAND HMI" %
%   B38:0/1  MAN_ADS_HTRS_ON  "COMMAND HMI" %

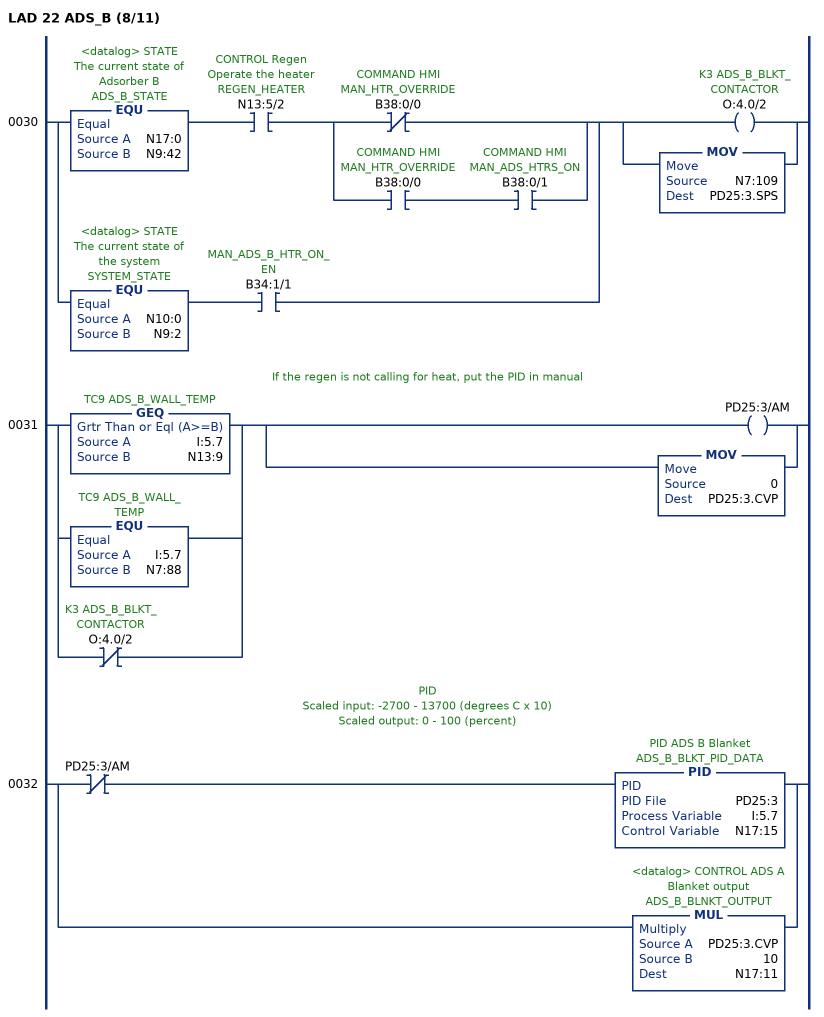
% Rung: 30 %
SOR BST EQU N17:0 N9:42 XIC N13:5/2 BST XIO B38:0/0 NXB XIC B38:0/0 XIC B38:0/1 BND NXB EQU N10:0 N9:2 XIC B34:1/1 BND BST OTE O:4.0/2 NXB MOV N7:109 PD25:3.SPS BND EOR
%   N17:0  ADS_B_STATE  "<datalog> STATE The current state of Adsorber B" %
%   N9:42  ADS_REGEN  "STATE ADS Regen" %
%   N13:5/2  REGEN_HEATER  "CONTROL Regen Operate the heater" %
%   B38:0/0  MAN_HTR_OVERRIDE  "COMMAND HMI" %
%   B38:0/1  MAN_ADS_HTRS_ON  "COMMAND HMI" %
%   N10:0  SYSTEM_STATE  "<datalog> STATE The current state of the system" %
%   N9:2  SYSTEM_MANUAL  "STATE System Manual" %
%   B34:1/1  MAN_ADS_B_HTR_ON_EN %
%   O:4.0/2  ADS_B_BLKT_CONTACTOR  "K3" %
%   N7:109  BLANKET_SP  "<datalog> ADS Blanket PID Setpoint" %
% Rung: 31 %
% If the regen is not calling for heat, put the PID in manual %
SOR BST GEQ I:5.7 N13:9 NXB EQU I:5.7 N7:88 NXB XIO O:4.0/2 BND BST OTE PD25:3/AM NXB MOV 0 PD25:3.CVP BND EOR
%   I:5.7  ADS_B_WALL_TEMP  "TC9" %
%   N13:9  BLANKET_LIMIT  "ADS Blanket Temp Limit" %
%   N7:88  TC_OPEN_SP  "CONFIG TC Open Setpoint" %
%   O:4.0/2  ADS_B_BLKT_CONTACTOR  "K3" %
% Rung: 32 %
% PID
% Scaled input: -2700 - 13700 (degrees C x 10)
% Scaled output: 0 - 100 (percent) %
SOR BST XIO PD25:3/AM PID PD25:3 I:5.7 N17:15 NXB MUL PD25:3.CVP 10 N17:11 BND EOR
%   PD25:3  ADS_B_BLKT_PID_DATA  "PID ADS B Blanket" %
%   I:5.7  ADS_B_WALL_TEMP  "TC9" %
%   N17:15  ADS_B_BLKT_OUTPT_RAW  "CONTROL ADS B Blanket PID Output Raw" %
%   N17:11  ADS_B_BLNKT_OUTPUT  "<datalog> CONTROL ADS A Blanket output" %

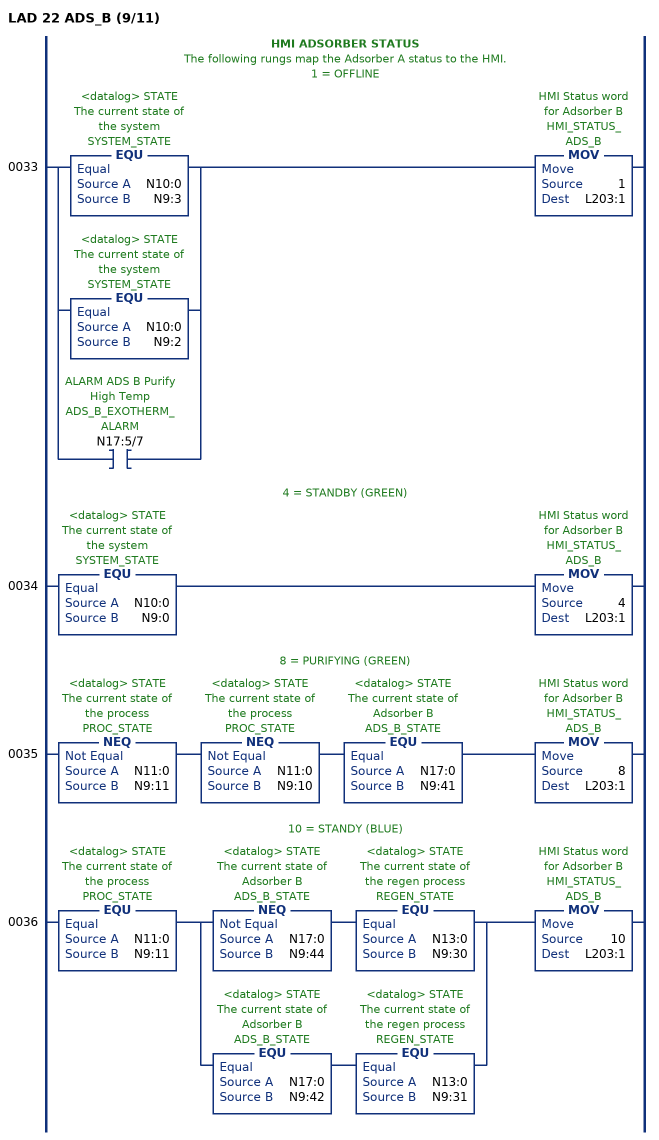
% Rung: 33 %
% TITLE: HMI ADSORBER STATUS %
% The following rungs map the Adsorber A status to the HMI.
% 1 = OFFLINE %
SOR BST EQU N10:0 N9:3 NXB EQU N10:0 N9:2 NXB XIC N17:5/7 BND MOV 1 L203:1 EOR
%   N10:0  SYSTEM_STATE  "<datalog> STATE The current state of the system" %
%   N9:3  SYSTEM_ALARM  "STATE System Alarm" %
%   N9:2  SYSTEM_MANUAL  "STATE System Manual" %
%   N17:5/7  ADS_B_EXOTHERM_ALARM  "ALARM ADS B Purify High Temp" %
%   L203:1  HMI_STATUS_ADS_B  "HMI Status word for Adsorber B" %
% Rung: 34 %
% 4 = STANDBY (GREEN) %
SOR EQU N10:0 N9:0 MOV 4 L203:1 EOR
%   N10:0  SYSTEM_STATE  "<datalog> STATE The current state of the system" %
%   N9:0  SYSTEM_STANDBY  "STATE System Standby" %
%   L203:1  HMI_STATUS_ADS_B  "HMI Status word for Adsorber B" %
% Rung: 35 %
% 8 = PURIFYING (GREEN) %
SOR NEQ N11:0 N9:11 NEQ N11:0 N9:10 EQU N17:0 N9:41 MOV 8 L203:1 EOR
%   N11:0  PROC_STATE  "<datalog> STATE The current state of the process" %
%   N9:11  PROC_REGEN_B  "STATE Process Regen B" %
%   N9:10  PROCESS_STANDBY  "STATE Process Standby" %
%   N17:0  ADS_B_STATE  "<datalog> STATE The current state of Adsorber B" %
%   N9:41  ADS_PURIFY  "STATE ADS Purify" %
%   L203:1  HMI_STATUS_ADS_B  "HMI Status word for Adsorber B" %
% Rung: 36 %
% 10 = STANDY (BLUE) %
SOR EQU N11:0 N9:11 BST NEQ N17:0 N9:44 EQU N13:0 N9:30 NXB EQU N17:0 N9:42 EQU N13:0 N9:31 BND MOV 10 L203:1 EOR
%   N11:0  PROC_STATE  "<datalog> STATE The current state of the process" %
%   N9:11  PROC_REGEN_B  "STATE Process Regen B" %
%   N17:0  ADS_B_STATE  "<datalog> STATE The current state of Adsorber B" %
%   N9:44  ADS_ALARM  "STATE ADS Alarm" %
%   N13:0  REGEN_STATE  "<datalog> STATE The current state of the regen process" %
%   N9:30  REGEN_STANDBY  "STATE Regen Standby" %
%   N9:42  ADS_REGEN  "STATE ADS Regen" %
%   N9:31  REGEN_DELAY  "STATE Regen Delay" %
%   L203:1  HMI_STATUS_ADS_B  "HMI Status word for Adsorber B" %

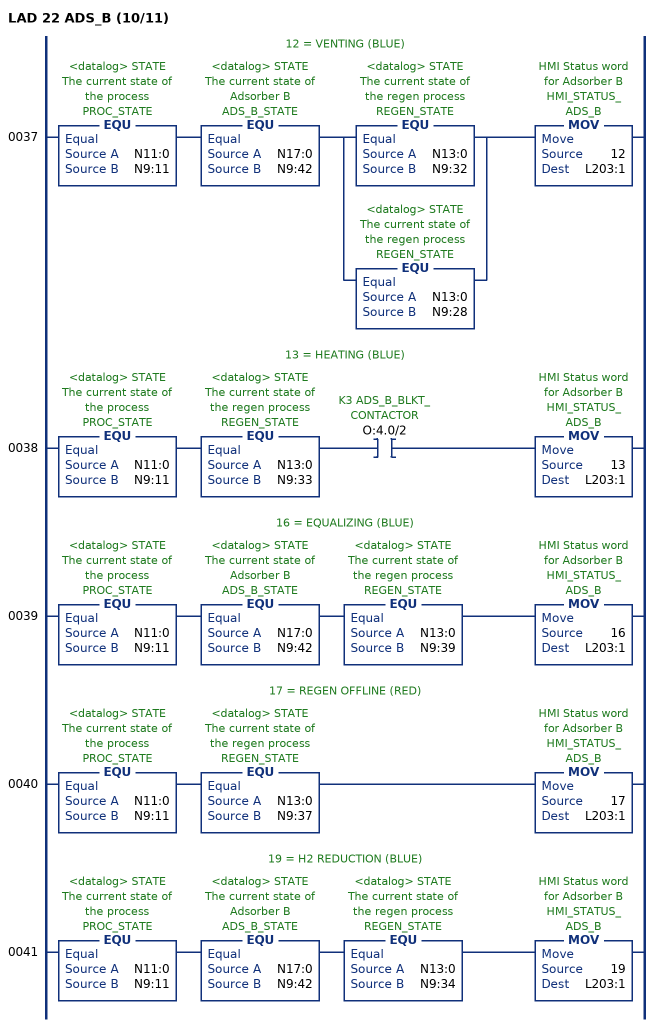
% Rung: 37 %
% 12 = VENTING (BLUE) %
SOR EQU N11:0 N9:11 EQU N17:0 N9:42 BST EQU N13:0 N9:32 NXB EQU N13:0 N9:28 BND MOV 12 L203:1 EOR
%   N11:0  PROC_STATE  "<datalog> STATE The current state of the process" %
%   N9:11  PROC_REGEN_B  "STATE Process Regen B" %
%   N17:0  ADS_B_STATE  "<datalog> STATE The current state of Adsorber B" %
%   N9:42  ADS_REGEN  "STATE ADS Regen" %
%   N13:0  REGEN_STATE  "<datalog> STATE The current state of the regen process" %
%   N9:32  REGEN_VENT  "STATE Regen Vent" %
%   N9:28  REGEN_VENT_2 %
%   L203:1  HMI_STATUS_ADS_B  "HMI Status word for Adsorber B" %
% Rung: 38 %
% 13 = HEATING (BLUE) %
SOR EQU N11:0 N9:11 EQU N13:0 N9:33 XIC O:4.0/2 MOV 13 L203:1 EOR
%   N11:0  PROC_STATE  "<datalog> STATE The current state of the process" %
%   N9:11  PROC_REGEN_B  "STATE Process Regen B" %
%   N13:0  REGEN_STATE  "<datalog> STATE The current state of the regen process" %
%   N9:33  REGEN_HEAT_BED  "STATE Regen Heat wall" %
%   O:4.0/2  ADS_B_BLKT_CONTACTOR  "K3" %
%   L203:1  HMI_STATUS_ADS_B  "HMI Status word for Adsorber B" %
% Rung: 39 %
% 16 = EQUALIZING (BLUE) %
SOR EQU N11:0 N9:11 EQU N17:0 N9:42 EQU N13:0 N9:39 MOV 16 L203:1 EOR
%   N11:0  PROC_STATE  "<datalog> STATE The current state of the process" %
%   N9:11  PROC_REGEN_B  "STATE Process Regen B" %
%   N17:0  ADS_B_STATE  "<datalog> STATE The current state of Adsorber B" %
%   N9:42  ADS_REGEN  "STATE ADS Regen" %
%   N13:0  REGEN_STATE  "<datalog> STATE The current state of the regen process" %
%   N9:39  REGEN_EQUALIZE  "STATE Regen Equalize" %
%   L203:1  HMI_STATUS_ADS_B  "HMI Status word for Adsorber B" %
% Rung: 40 %
% 17 = REGEN OFFLINE (RED) %
SOR EQU N11:0 N9:11 EQU N13:0 N9:37 MOV 17 L203:1 EOR
%   N11:0  PROC_STATE  "<datalog> STATE The current state of the process" %
%   N9:11  PROC_REGEN_B  "STATE Process Regen B" %
%   N13:0  REGEN_STATE  "<datalog> STATE The current state of the regen process" %
%   N9:37  REGEN_ALARM  "STATE Regen Alarm" %
%   L203:1  HMI_STATUS_ADS_B  "HMI Status word for Adsorber B" %
% Rung: 41 %
% 19 = H2 REDUCTION (BLUE) %
SOR EQU N11:0 N9:11 EQU N17:0 N9:42 EQU N13:0 N9:34 MOV 19 L203:1 EOR
%   N11:0  PROC_STATE  "<datalog> STATE The current state of the process" %
%   N9:11  PROC_REGEN_B  "STATE Process Regen B" %
%   N17:0  ADS_B_STATE  "<datalog> STATE The current state of Adsorber B" %
%   N9:42  ADS_REGEN  "STATE ADS Regen" %
%   N13:0  REGEN_STATE  "<datalog> STATE The current state of the regen process" %
%   N9:34  REGEN_H2_REDUCTION  "STATE Regen Running" %
%   L203:1  HMI_STATUS_ADS_B  "HMI Status word for Adsorber B" %

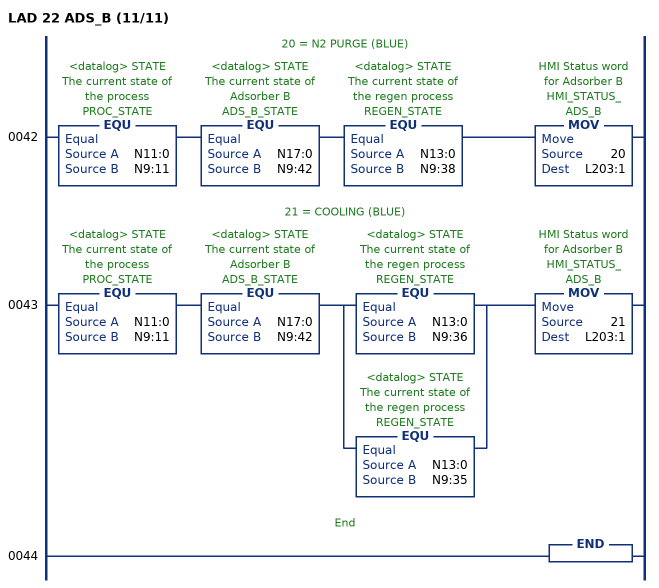
% Rung: 42 %
% 20 = N2 PURGE (BLUE) %
SOR EQU N11:0 N9:11 EQU N17:0 N9:42 EQU N13:0 N9:38 MOV 20 L203:1 EOR
%   N11:0  PROC_STATE  "<datalog> STATE The current state of the process" %
%   N9:11  PROC_REGEN_B  "STATE Process Regen B" %
%   N17:0  ADS_B_STATE  "<datalog> STATE The current state of Adsorber B" %
%   N9:42  ADS_REGEN  "STATE ADS Regen" %
%   N13:0  REGEN_STATE  "<datalog> STATE The current state of the regen process" %
%   N9:38  REGEN_PURGE  "STATE Regen Hot Purge" %
%   L203:1  HMI_STATUS_ADS_B  "HMI Status word for Adsorber B" %
% Rung: 43 %
% 21 = COOLING (BLUE) %
SOR EQU N11:0 N9:11 EQU N17:0 N9:42 BST EQU N13:0 N9:36 NXB EQU N13:0 N9:35 BND MOV 21 L203:1 EOR
%   N11:0  PROC_STATE  "<datalog> STATE The current state of the process" %
%   N9:11  PROC_REGEN_B  "STATE Process Regen B" %
%   N17:0  ADS_B_STATE  "<datalog> STATE The current state of Adsorber B" %
%   N9:42  ADS_REGEN  "STATE ADS Regen" %
%   N13:0  REGEN_STATE  "<datalog> STATE The current state of the regen process" %
%   N9:36  REGEN_COOL  "STATE Regen Cool" %
%   N9:35  REGEN_COOL_WALL  "STATE Regen Cool wall" %
%   L203:1  HMI_STATUS_ADS_B  "HMI Status word for Adsorber B" %
% Rung: 44 %
% End %
SOR END EOR

LADDER 23 "ADS_B_FLT"    % Controls the Adsorber B faults %
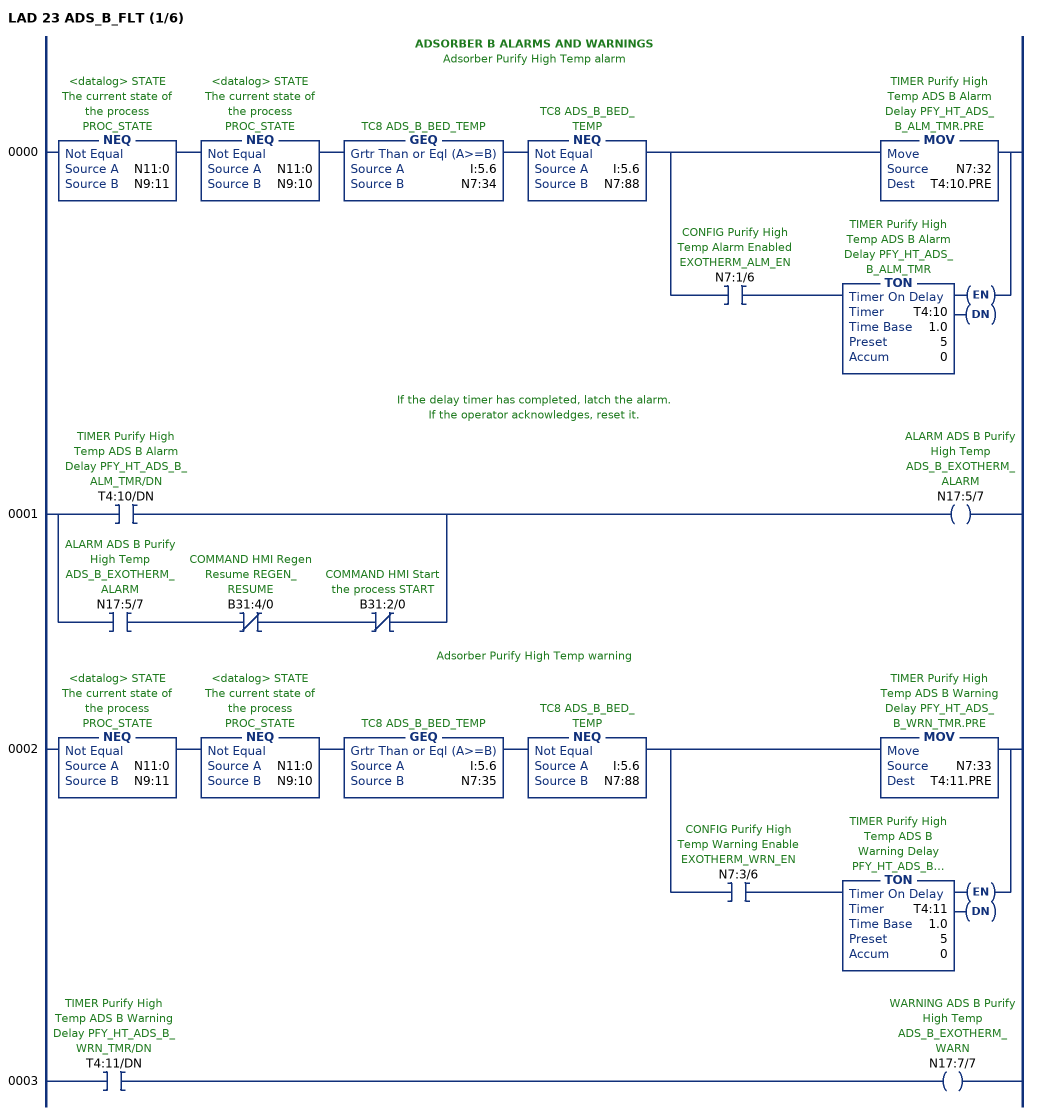
% Rung: 0 %
% TITLE: ADSORBER B ALARMS AND WARNINGS %
% Adsorber Purify High Temp alarm %
SOR NEQ N11:0 N9:11 NEQ N11:0 N9:10 GEQ I:5.6 N7:34 NEQ I:5.6 N7:88 BST MOV N7:32 T4:10.PRE NXB XIC N7:1/6 TON T4:10 1.0 5 0 BND EOR
%   N11:0  PROC_STATE  "<datalog> STATE The current state of the process" %
%   N9:11  PROC_REGEN_B  "STATE Process Regen B" %
%   N9:10  PROCESS_STANDBY  "STATE Process Standby" %
%   I:5.6  ADS_B_BED_TEMP  "TC8" %
%   N7:34  EXOTHERM_ALM_SP  "CONFIG Purify High Temp Alarm Setpoint" %
%   N7:88  TC_OPEN_SP  "CONFIG TC Open Setpoint" %
%   N7:32  EXOTHERM_ALM_DLY  "CONFIG Purify High Temp Alarm Delay" %
%   T4:10  PFY_HT_ADS_B_ALM_TMR  "TIMER Purify High Temp ADS B Alarm Delay" %
%   N7:1/6  EXOTHERM_ALM_EN  "CONFIG Purify High Temp Alarm Enabled" %
% Rung: 1 %
% If the delay timer has completed, latch the alarm.
% If the operator acknowledges, reset it. %
SOR BST XIC T4:10/DN NXB XIC N17:5/7 XIO B31:4/0 XIO B31:2/0 BND OTE N17:5/7 EOR
%   T4:10  PFY_HT_ADS_B_ALM_TMR  "TIMER Purify High Temp ADS B Alarm Delay" %
%   N17:5/7  ADS_B_EXOTHERM_ALARM  "ALARM ADS B Purify High Temp" %
%   B31:4/0  REGEN_RESUME  "COMMAND HMI Regen Resume" %
%   B31:2/0  START  "COMMAND HMI Start the process" %
% Rung: 2 %
% Adsorber Purify High Temp warning %
SOR NEQ N11:0 N9:11 NEQ N11:0 N9:10 GEQ I:5.6 N7:35 NEQ I:5.6 N7:88 BST MOV N7:33 T4:11.PRE NXB XIC N7:3/6 TON T4:11 1.0 5 0 BND EOR
%   N11:0  PROC_STATE  "<datalog> STATE The current state of the process" %
%   N9:11  PROC_REGEN_B  "STATE Process Regen B" %
%   N9:10  PROCESS_STANDBY  "STATE Process Standby" %
%   I:5.6  ADS_B_BED_TEMP  "TC8" %
%   N7:35  EXOTHERM_WRN_SP  "CONFIG Purify High Temp Warning Setpoint" %
%   N7:88  TC_OPEN_SP  "CONFIG TC Open Setpoint" %
%   N7:33  EXOTHERM_WRN_DLY  "CONFIG Purify High Temp Warning Delay" %
%   T4:11  PFY_HT_ADS_B_WRN_TMR  "TIMER Purify High Temp ADS B Warning Delay" %
%   N7:3/6  EXOTHERM_WRN_EN  "CONFIG Purify High Temp Warning Enable" %
% Rung: 3 %
SOR XIC T4:11/DN OTE N17:7/7 EOR
%   T4:11  PFY_HT_ADS_B_WRN_TMR  "TIMER Purify High Temp ADS B Warning Delay" %
%   N17:7/7  ADS_B_EXOTHERM_WARN  "WARNING ADS B Purify High Temp" %

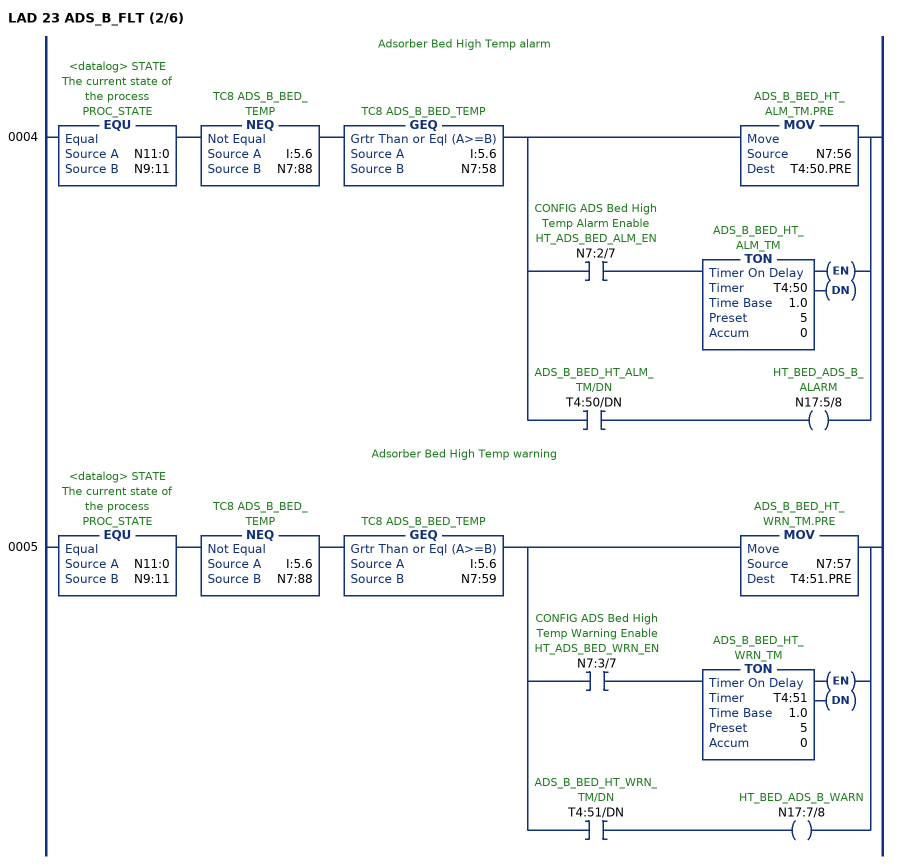
% Rung: 4 %
% Adsorber Bed High Temp alarm %
SOR EQU N11:0 N9:11 NEQ I:5.6 N7:88 GEQ I:5.6 N7:58 BST MOV N7:56 T4:50.PRE NXB XIC N7:2/7 TON T4:50 1.0 5 0 NXB XIC T4:50/DN OTE N17:5/8 BND EOR
%   N11:0  PROC_STATE  "<datalog> STATE The current state of the process" %
%   N9:11  PROC_REGEN_B  "STATE Process Regen B" %
%   I:5.6  ADS_B_BED_TEMP  "TC8" %
%   N7:88  TC_OPEN_SP  "CONFIG TC Open Setpoint" %
%   N7:58  HT_ADS_BED_ALM_SP  "CONFIG ADS Bed High Temp Alarm Setpoint" %
%   N7:56  HT_ADS_BED_ALM_DLY  "CONFIG ADS Bed High Temp Alarm Delay" %
%   T4:50  ADS_B_BED_HT_ALM_TM %
%   N7:2/7  HT_ADS_BED_ALM_EN  "CONFIG ADS Bed High Temp Alarm Enable" %
%   N17:5/8  HT_BED_ADS_B_ALARM %
% Rung: 5 %
% Adsorber Bed High Temp warning %
SOR EQU N11:0 N9:11 NEQ I:5.6 N7:88 GEQ I:5.6 N7:59 BST MOV N7:57 T4:51.PRE NXB XIC N7:3/7 TON T4:51 1.0 5 0 NXB XIC T4:51/DN OTE N17:7/8 BND EOR
%   N11:0  PROC_STATE  "<datalog> STATE The current state of the process" %
%   N9:11  PROC_REGEN_B  "STATE Process Regen B" %
%   I:5.6  ADS_B_BED_TEMP  "TC8" %
%   N7:88  TC_OPEN_SP  "CONFIG TC Open Setpoint" %
%   N7:59  HT_ADS_BED_WRN_SP  "CONFIG ADS Bed High Temp Warning Setpoint" %
%   N7:57  HT_ADS_BED_WRN_DLY  "CONFIG ADS Bed High Temp Warning Delay" %
%   T4:51  ADS_B_BED_HT_WRN_TM %
%   N7:3/7  HT_ADS_BED_WRN_EN  "CONFIG ADS Bed High Temp Warning Enable" %
%   N17:7/8  HT_BED_ADS_B_WARN %

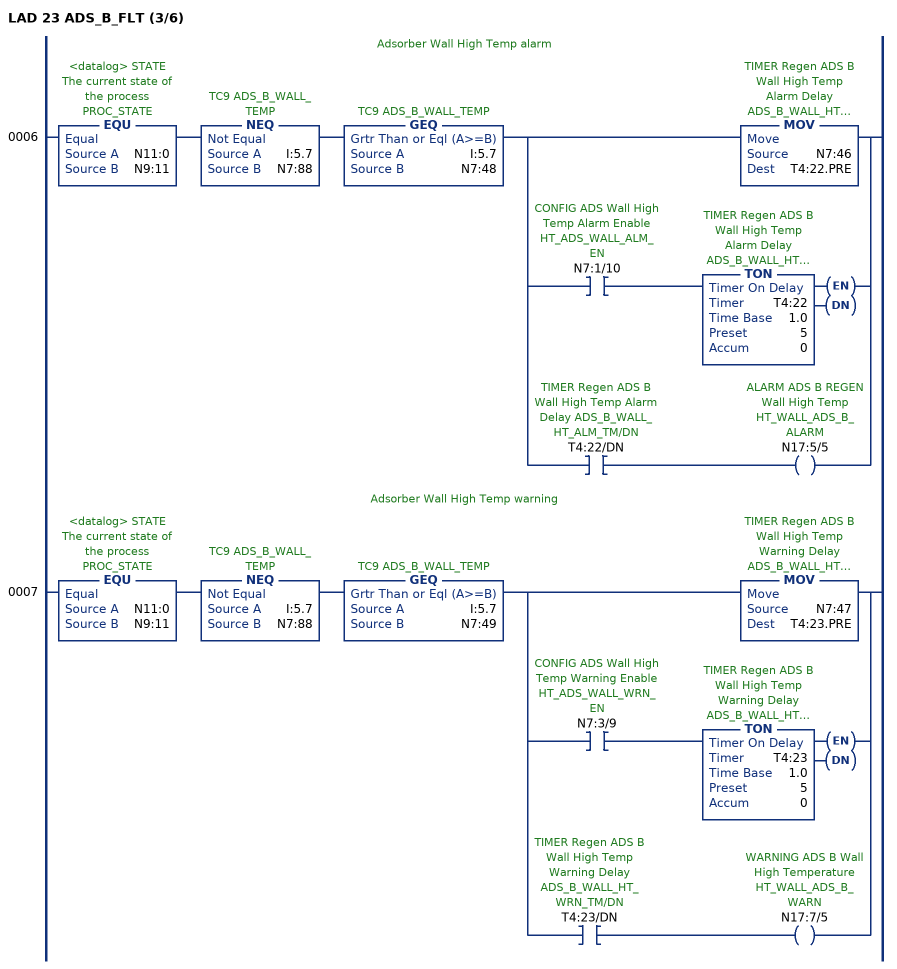
% Rung: 6 %
% Adsorber Wall High Temp alarm %
SOR EQU N11:0 N9:11 NEQ I:5.7 N7:88 GEQ I:5.7 N7:48 BST MOV N7:46 T4:22.PRE NXB XIC N7:1/10 TON T4:22 1.0 5 0 NXB XIC T4:22/DN OTE N17:5/5 BND EOR
%   N11:0  PROC_STATE  "<datalog> STATE The current state of the process" %
%   N9:11  PROC_REGEN_B  "STATE Process Regen B" %
%   I:5.7  ADS_B_WALL_TEMP  "TC9" %
%   N7:88  TC_OPEN_SP  "CONFIG TC Open Setpoint" %
%   N7:48  HT_ADS_WALL_ALM_SP  "CONFIG ADS Wall High Temp Alarm Setpoint" %
%   N7:46  HT_ADS_WALL_ALM_DLY  "CONFIG ADS Wall High Temp Alarm Delay" %
%   T4:22  ADS_B_WALL_HT_ALM_TM  "TIMER Regen ADS B Wall High Temp Alarm Delay" %
%   N7:1/10  HT_ADS_WALL_ALM_EN  "CONFIG ADS Wall High Temp Alarm Enable" %
%   N17:5/5  HT_WALL_ADS_B_ALARM  "ALARM ADS B REGEN Wall High Temp" %
% Rung: 7 %
% Adsorber Wall High Temp warning %
SOR EQU N11:0 N9:11 NEQ I:5.7 N7:88 GEQ I:5.7 N7:49 BST MOV N7:47 T4:23.PRE NXB XIC N7:3/9 TON T4:23 1.0 5 0 NXB XIC T4:23/DN OTE N17:7/5 BND EOR
%   N11:0  PROC_STATE  "<datalog> STATE The current state of the process" %
%   N9:11  PROC_REGEN_B  "STATE Process Regen B" %
%   I:5.7  ADS_B_WALL_TEMP  "TC9" %
%   N7:88  TC_OPEN_SP  "CONFIG TC Open Setpoint" %
%   N7:49  HT_ADS_WALL_WRN_SP  "CONFIG ADS Wall High Temp Warning Setpoint" %
%   N7:47  HT_ADS_WALL_WRN_DLY  "CONFIG ADS Wall High Temp Warning Delay" %
%   T4:23  ADS_B_WALL_HT_WRN_TM  "TIMER Regen ADS B Wall High Temp Warning Delay" %
%   N7:3/9  HT_ADS_WALL_WRN_EN  "CONFIG ADS Wall High Temp Warning Enable" %
%   N17:7/5  HT_WALL_ADS_B_WARN  "WARNING ADS B Wall High Temperature" %

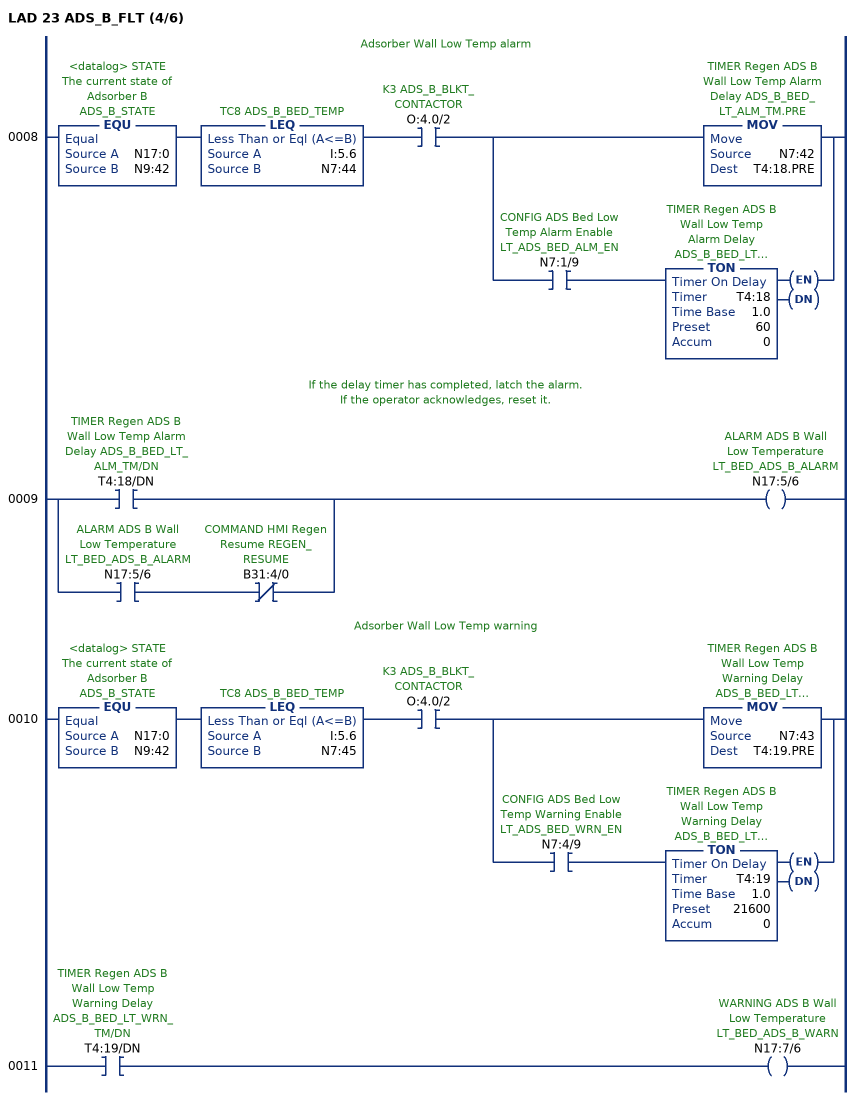
% Rung: 8 %
% Adsorber Wall Low Temp alarm %
SOR EQU N17:0 N9:42 LEQ I:5.6 N7:44 XIC O:4.0/2 BST MOV N7:42 T4:18.PRE NXB XIC N7:1/9 TON T4:18 1.0 60 0 BND EOR
%   N17:0  ADS_B_STATE  "<datalog> STATE The current state of Adsorber B" %
%   N9:42  ADS_REGEN  "STATE ADS Regen" %
%   I:5.6  ADS_B_BED_TEMP  "TC8" %
%   N7:44  LT_ADS_BED_ALM_SP  "CONFIG ADS Bed Low Temp Alarm Setpoint" %
%   O:4.0/2  ADS_B_BLKT_CONTACTOR  "K3" %
%   N7:42  LT_ADS_BED_ALM_DLY  "CONFIG ADS Bed Low Temp Alarm Delay" %
%   T4:18  ADS_B_BED_LT_ALM_TM  "TIMER Regen ADS B Wall Low Temp Alarm Delay" %
%   N7:1/9  LT_ADS_BED_ALM_EN  "CONFIG ADS Bed Low Temp Alarm Enable" %
% Rung: 9 %
% If the delay timer has completed, latch the alarm.
% If the operator acknowledges, reset it. %
SOR BST XIC T4:18/DN NXB XIC N17:5/6 XIO B31:4/0 BND OTE N17:5/6 EOR
%   T4:18  ADS_B_BED_LT_ALM_TM  "TIMER Regen ADS B Wall Low Temp Alarm Delay" %
%   N17:5/6  LT_BED_ADS_B_ALARM  "ALARM ADS B Wall Low Temperature" %
%   B31:4/0  REGEN_RESUME  "COMMAND HMI Regen Resume" %
% Rung: 10 %
% Adsorber Wall Low Temp warning %
SOR EQU N17:0 N9:42 LEQ I:5.6 N7:45 XIC O:4.0/2 BST MOV N7:43 T4:19.PRE NXB XIC N7:4/9 TON T4:19 1.0 21600 0 BND EOR
%   N17:0  ADS_B_STATE  "<datalog> STATE The current state of Adsorber B" %
%   N9:42  ADS_REGEN  "STATE ADS Regen" %
%   I:5.6  ADS_B_BED_TEMP  "TC8" %
%   N7:45  LT_ADS_BED_WRN_SP  "CONFIG ADS Bed Low Temp Warning Setpoint" %
%   O:4.0/2  ADS_B_BLKT_CONTACTOR  "K3" %
%   N7:43  LT_ADS_BED_WRN_DLY  "CONFIG ADS Bed Low Temp Warning Delay" %
%   T4:19  ADS_B_BED_LT_WRN_TM  "TIMER Regen ADS B Wall Low Temp Warning Delay" %
%   N7:4/9  LT_ADS_BED_WRN_EN  "CONFIG ADS Bed Low Temp Warning Enable" %
% Rung: 11 %
SOR XIC T4:19/DN OTE N17:7/6 EOR
%   T4:19  ADS_B_BED_LT_WRN_TM  "TIMER Regen ADS B Wall Low Temp Warning Delay" %
%   N17:7/6  LT_BED_ADS_B_WARN  "WARNING ADS B Wall Low Temperature" %

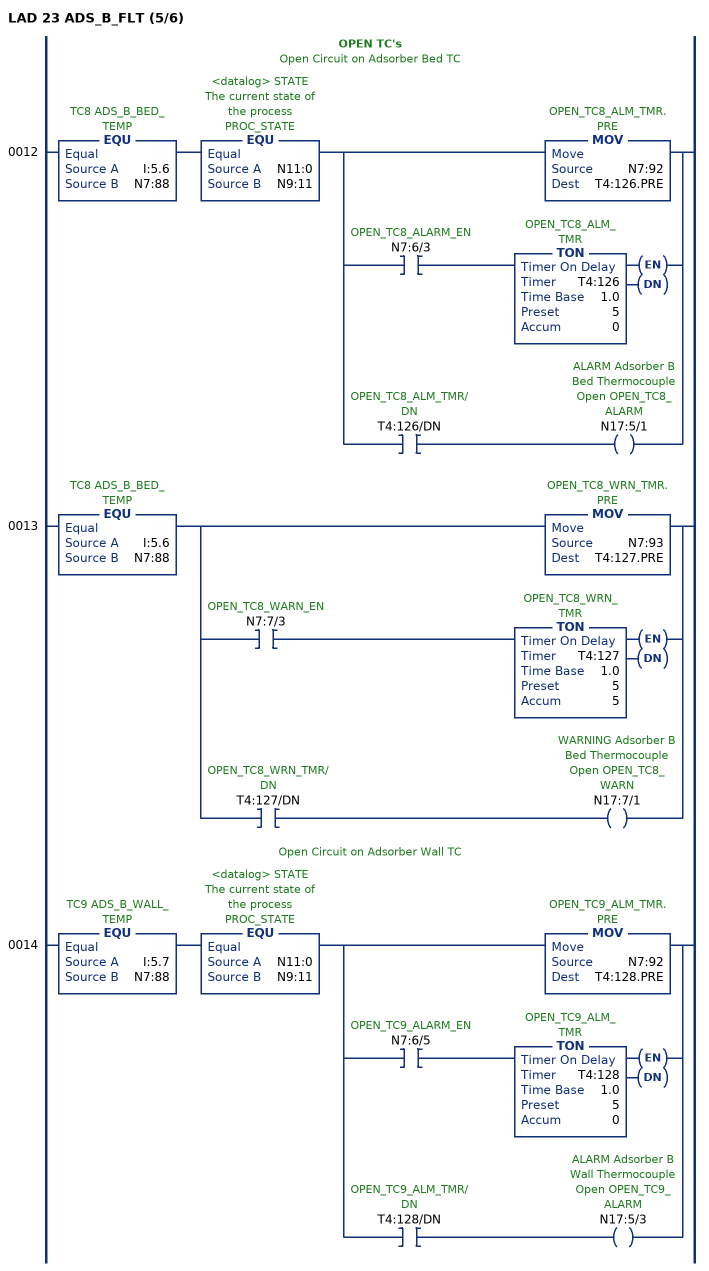
% Rung: 12 %
% TITLE: OPEN TC's %
% Open Circuit on Adsorber Bed TC %
SOR EQU I:5.6 N7:88 EQU N11:0 N9:11 BST MOV N7:92 T4:126.PRE NXB XIC N7:6/3 TON T4:126 1.0 5 0 NXB XIC T4:126/DN OTE N17:5/1 BND EOR
%   I:5.6  ADS_B_BED_TEMP  "TC8" %
%   N7:88  TC_OPEN_SP  "CONFIG TC Open Setpoint" %
%   N11:0  PROC_STATE  "<datalog> STATE The current state of the process" %
%   N9:11  PROC_REGEN_B  "STATE Process Regen B" %
%   N7:92  OPEN_TC_ALM_DLY  "CONFIG TC Open Alarm Delay" %
%   T4:126  OPEN_TC8_ALM_TMR %
%   N7:6/3  OPEN_TC8_ALARM_EN %
%   N17:5/1  OPEN_TC8_ALARM  "ALARM Adsorber B Bed Thermocouple Open" %
% Rung: 13 %
SOR EQU I:5.6 N7:88 BST MOV N7:93 T4:127.PRE NXB XIC N7:7/3 TON T4:127 1.0 5 5 NXB XIC T4:127/DN OTE N17:7/1 BND EOR
%   I:5.6  ADS_B_BED_TEMP  "TC8" %
%   N7:88  TC_OPEN_SP  "CONFIG TC Open Setpoint" %
%   N7:93  OPEN_TC_WRN_DLY  "CONFIG TC Open Warning Delay" %
%   T4:127  OPEN_TC8_WRN_TMR %
%   N7:7/3  OPEN_TC8_WARN_EN %
%   N17:7/1  OPEN_TC8_WARN  "WARNING Adsorber B Bed Thermocouple Open" %
% Rung: 14 %
% Open Circuit on Adsorber Wall TC %
SOR EQU I:5.7 N7:88 EQU N11:0 N9:11 BST MOV N7:92 T4:128.PRE NXB XIC N7:6/5 TON T4:128 1.0 5 0 NXB XIC T4:128/DN OTE N17:5/3 BND EOR
%   I:5.7  ADS_B_WALL_TEMP  "TC9" %
%   N7:88  TC_OPEN_SP  "CONFIG TC Open Setpoint" %
%   N11:0  PROC_STATE  "<datalog> STATE The current state of the process" %
%   N9:11  PROC_REGEN_B  "STATE Process Regen B" %
%   N7:92  OPEN_TC_ALM_DLY  "CONFIG TC Open Alarm Delay" %
%   T4:128  OPEN_TC9_ALM_TMR %
%   N7:6/5  OPEN_TC9_ALARM_EN %
%   N17:5/3  OPEN_TC9_ALARM  "ALARM Adsorber B Wall Thermocouple Open" %

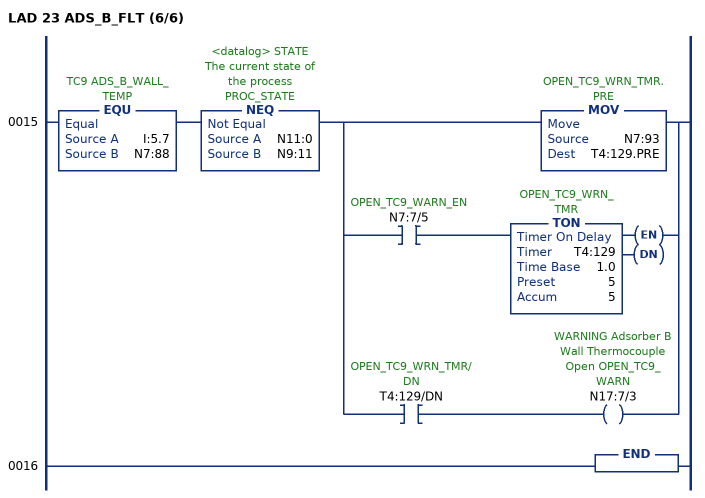
% Rung: 15 %
SOR EQU I:5.7 N7:88 NEQ N11:0 N9:11 BST MOV N7:93 T4:129.PRE NXB XIC N7:7/5 TON T4:129 1.0 5 5 NXB XIC T4:129/DN OTE N17:7/3 BND EOR
%   I:5.7  ADS_B_WALL_TEMP  "TC9" %
%   N7:88  TC_OPEN_SP  "CONFIG TC Open Setpoint" %
%   N11:0  PROC_STATE  "<datalog> STATE The current state of the process" %
%   N9:11  PROC_REGEN_B  "STATE Process Regen B" %
%   N7:93  OPEN_TC_WRN_DLY  "CONFIG TC Open Warning Delay" %
%   T4:129  OPEN_TC9_WRN_TMR %
%   N7:7/5  OPEN_TC9_WARN_EN %
%   N17:7/3  OPEN_TC9_WARN  "WARNING Adsorber B Wall Thermocouple Open" %
% Rung: 16 %
SOR END EOR

LADDER 24 "PREHEATER"
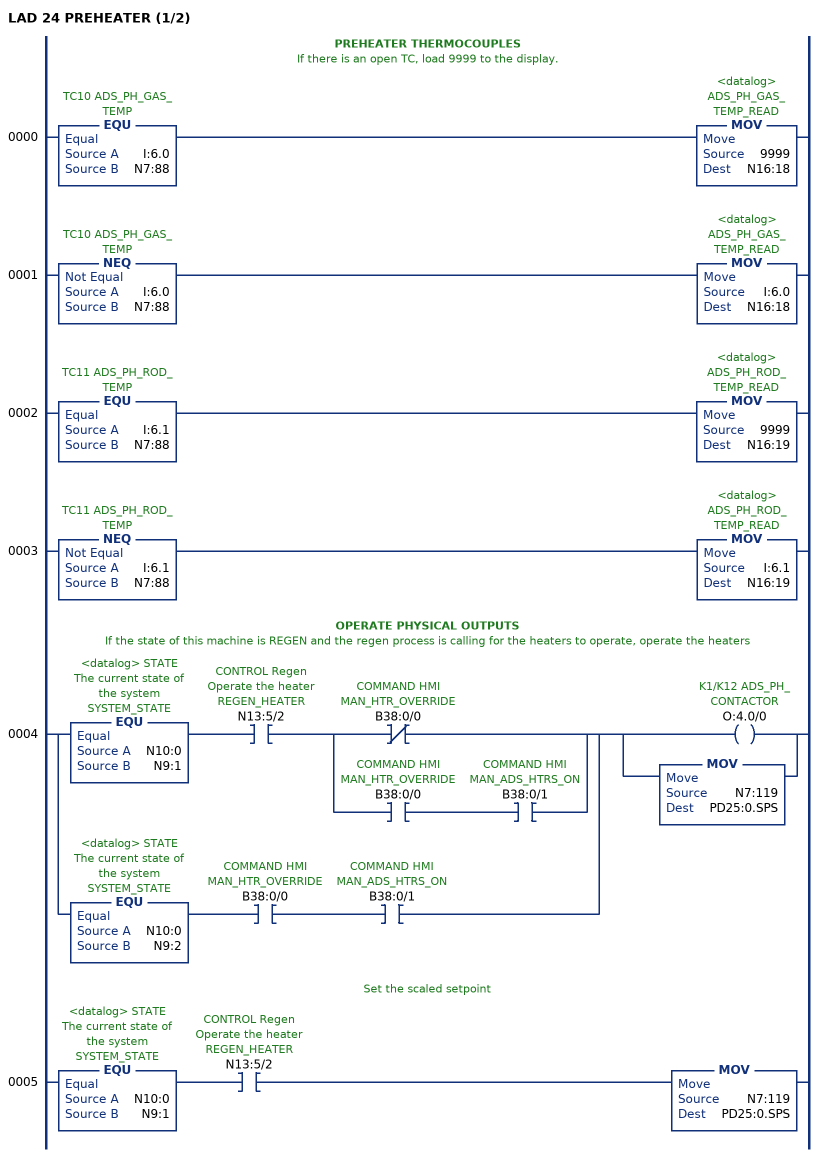
% Rung: 0 %
% TITLE: PREHEATER THERMOCOUPLES %
% If there is an open TC, load 9999 to the display. %
SOR EQU I:6.0 N7:88 MOV 9999 N16:18 EOR
%   I:6.0  ADS_PH_GAS_TEMP  "TC10" %
%   N7:88  TC_OPEN_SP  "CONFIG TC Open Setpoint" %
%   N16:18  ADS_PH_GAS_TEMP_READ  "<datalog>" %
% Rung: 1 %
SOR NEQ I:6.0 N7:88 MOV I:6.0 N16:18 EOR
%   I:6.0  ADS_PH_GAS_TEMP  "TC10" %
%   N7:88  TC_OPEN_SP  "CONFIG TC Open Setpoint" %
%   N16:18  ADS_PH_GAS_TEMP_READ  "<datalog>" %
% Rung: 2 %
SOR EQU I:6.1 N7:88 MOV 9999 N16:19 EOR
%   I:6.1  ADS_PH_ROD_TEMP  "TC11" %
%   N7:88  TC_OPEN_SP  "CONFIG TC Open Setpoint" %
%   N16:19  ADS_PH_ROD_TEMP_READ  "<datalog>" %
% Rung: 3 %
SOR NEQ I:6.1 N7:88 MOV I:6.1 N16:19 EOR
%   I:6.1  ADS_PH_ROD_TEMP  "TC11" %
%   N7:88  TC_OPEN_SP  "CONFIG TC Open Setpoint" %
%   N16:19  ADS_PH_ROD_TEMP_READ  "<datalog>" %
% Rung: 4 %
% TITLE: OPERATE PHYSICAL OUTPUTS %
% If the state of this machine is REGEN and the regen process is calling for the heaters to operate, operate the heaters %
SOR BST EQU N10:0 N9:1 XIC N13:5/2 BST XIO B38:0/0 NXB XIC B38:0/0 XIC B38:0/1 BND NXB EQU N10:0 N9:2 XIC B38:0/0 XIC B38:0/1 BND BST OTE O:4.0/0 NXB MOV N7:119 PD25:0.SPS BND EOR
%   N10:0  SYSTEM_STATE  "<datalog> STATE The current state of the system" %
%   N9:1  SYSTEM_PROCESS  "STATE System Process" %
%   N13:5/2  REGEN_HEATER  "CONTROL Regen Operate the heater" %
%   B38:0/0  MAN_HTR_OVERRIDE  "COMMAND HMI" %
%   B38:0/1  MAN_ADS_HTRS_ON  "COMMAND HMI" %
%   N9:2  SYSTEM_MANUAL  "STATE System Manual" %
%   O:4.0/0  ADS_PH_CONTACTOR  "K1/K12" %
%   N7:119  PREHEATER_SP  "<datalog> ADS Preheater PID Setpoint" %
% Rung: 5 %
% Set the scaled setpoint %
SOR EQU N10:0 N9:1 XIC N13:5/2 MOV N7:119 PD25:0.SPS EOR
%   N10:0  SYSTEM_STATE  "<datalog> STATE The current state of the system" %
%   N9:1  SYSTEM_PROCESS  "STATE System Process" %
%   N13:5/2  REGEN_HEATER  "CONTROL Regen Operate the heater" %
%   N7:119  PREHEATER_SP  "<datalog> ADS Preheater PID Setpoint" %

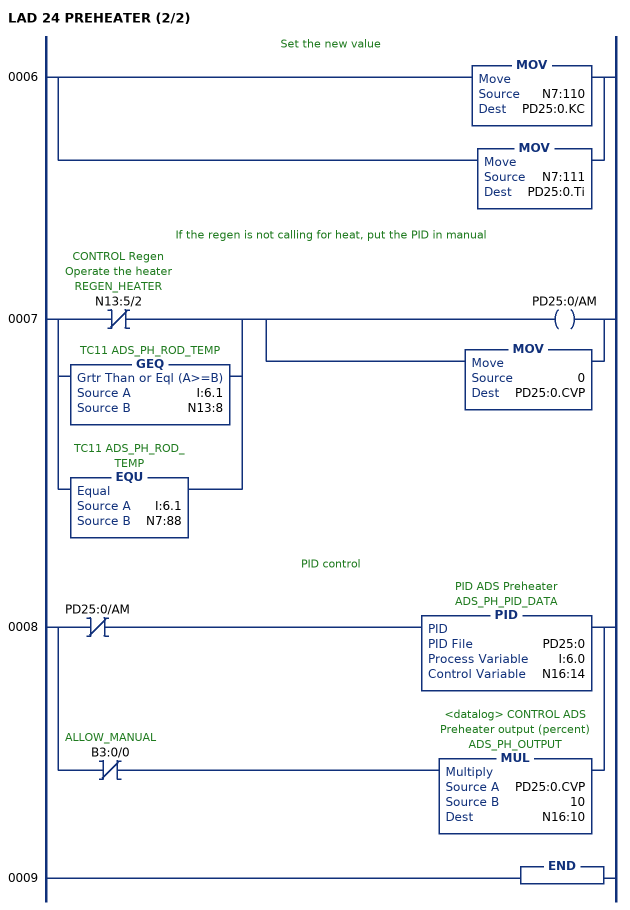
% Rung: 6 %
% Set the new value %
SOR BST MOV N7:110 PD25:0.KC NXB MOV N7:111 PD25:0.Ti BND EOR
%   N7:110  PREHEATER_P  "CONFIG Preheater Proportional Gain" %
%   N7:111  PREHEATER_I  "CONFIG Preheater Integral Gain" %
% Rung: 7 %
% If the regen is not calling for heat, put the PID in manual %
SOR BST XIO N13:5/2 NXB GEQ I:6.1 N13:8 NXB EQU I:6.1 N7:88 BND BST OTE PD25:0/AM NXB MOV 0 PD25:0.CVP BND EOR
%   N13:5/2  REGEN_HEATER  "CONTROL Regen Operate the heater" %
%   I:6.1  ADS_PH_ROD_TEMP  "TC11" %
%   N13:8  PH_ROD_LIMIT  "ADS Preheater Rod Temp Limit" %
%   N7:88  TC_OPEN_SP  "CONFIG TC Open Setpoint" %
% Rung: 8 %
% PID control %
SOR BST XIO PD25:0/AM PID PD25:0 I:6.0 N16:14 NXB XIO B3:0/0 MUL PD25:0.CVP 10 N16:10 BND EOR
%   PD25:0  ADS_PH_PID_DATA  "PID ADS Preheater" %
%   I:6.0  ADS_PH_GAS_TEMP  "TC10" %
%   N16:14  ADS_PH_OUTPUT_RAW  "CONTROL ADS A Preheater PID Output Raw" %
%   B3:0/0  ALLOW_MANUAL %
%   N16:10  ADS_PH_OUTPUT  "<datalog> CONTROL ADS Preheater output (percent)" %
% Rung: 9 %
SOR END EOR

LADDER 25 "PH_FLT"
